LIN {X 0,Y 162.947,Z 318.354,A -85,B 0,C 180,E1 -26149.316,E2 -26149.316} C_VEL
LIN {X 0,Y 160.484,Z 333.964,A -85,B 0,C 180,E1 -26150.172,E2 -26150.172} C_VEL
LIN {X 0,Y 157.007,Z 349.23,A -85,B 0,C 180,E1 -26151.399,E2 -26151.399} C_VEL
LIN {X 0,Y 152.992,Z 362.96,A -85,B 0,C 180,E1 -26152.919,E2 -26152.919} C_VEL
LIN {X 0,Y 148.184,Z 376.471,A -85,B 0,C 180,E1 -26154.895,E2 -26154.895} C_VEL
LIN {X 0,Y 142.969,Z 388.947,A -85,B 0,C 180,E1 -26157.265,E2 -26157.265} C_VEL
LIN {X 0,Y 137.361,Z 400.576,A -85,B 0,C 180,E1 -26160.074,E2 -26160.074} C_VEL
LIN {X 0,Y 131.045,Z 412.295,A -85,B 0,C 180,E1 -26163.738,E2 -26163.738} C_VEL
LIN {X 0,Y 125.325,Z 422.137,A -85,B 0,C 180,E1 -26167.756,E2 -26167.756} C_VEL
LIN {X 0,Y 119.407,Z 431.78,A -85,B 0,C 180,E1 -26172.884,E2 -26172.884} C_VEL
LIN {X 0,Y 115.037,Z 438.966,A -85,B 0,C 180,E1 -26177.828,E2 -26177.828} C_VEL
LIN {X 0,Y 110.501,Z 446.462,A -85,B 0,C 180,E1 -26184.524,E2 -26184.524} C_VEL
LIN {X 0,Y 107.298,Z 452.585,A -85,B 0,C 180,E1 -26191.875,E2 -26191.875} C_VEL
LIN {X 0,Y 105.639,Z 456.228,A -85,B 0,C 180,E1 -26197.645,E2 -26197.645} C_VEL
LIN {X 0,Y 104.586,Z 459.955,A -85,B 0,C 180,E1 -26205.591,E2 -26205.591} C_VEL
LIN {X 0,Y 104.541,Z 461.374,A -85,B 0,C 180,E1 -26209.743,E2 -26209.743} C_VEL
LIN {X 0,Y 105.346,Z 463.187,A -85,B 0,C 180,E1 -26217.838,E2 -26217.838} C_VEL
LIN {X 0,Y 107.662,Z 463.763,A -85,B 0,C 180,E1 -26225.978,E2 -26225.978} C_VEL
LIN {X 0,Y 111.789,Z 463.039,A -85,B 0,C 180,E1 -26233.751,E2 -26233.751} C_VEL
LIN {X 0,Y 117.628,Z 460.978,A -85,B 0,C 180,E1 -26240.959,E2 -26240.959} C_VEL
LIN {X 0,Y 125.074,Z 457.514,A -85,B 0,C 180,E1 -26247.441,E2 -26247.441} C_VEL
LIN {X 0,Y 133.883,Z 452.565,A -85,B 0,C 180,E1 -26253.173,E2 -26253.173} C_VEL
LIN {X 0,Y 143.854,Z 445.982,A -85,B 0,C 180,E1 -26258.161,E2 -26258.161} C_VEL
LIN {X 0,Y 152.435,Z 439.533,A -85,B 0,C 180,E1 -26261.583,E2 -26261.583} C_VEL
LIN {X 0,Y 162.624,Z 430.726,A -85,B 0,C 180,E1 -26264.971,E2 -26264.971} C_VEL
LIN {X 0,Y 172.579,Z 420.723,A -85,B 0,C 180,E1 -26267.781,E2 -26267.781} C_VEL
LIN {X 0,Y 181.957,Z 409.798,A -85,B 0,C 180,E1 -26270.035,E2 -26270.035} C_VEL
LIN {X 0,Y 190.529,Z 398.113,A -85,B 0,C 180,E1 -26271.871,E2 -26271.871} C_VEL
LIN {X 0,Y 198.109,Z 385.919,A -85,B 0,C 180,E1 -26273.364,E2 -26273.364} C_VEL
LIN {X 0,Y 204.736,Z 373.274,A -85,B 0,C 180,E1 -26274.55,E2 -26274.55} C_VEL
LIN {X 0,Y 211.024,Z 358.642,A -85,B 0,C 180,E1 -26275.59,E2 -26275.59} C_VEL
LIN {X 0,Y 215.218,Z 346.337,A -85,B 0,C 180,E1 -26276.255,E2 -26276.255} C_VEL
LIN {X 0,Y 219.141,Z 331.367,A -85,B 0,C 180,E1 -26276.858,E2 -26276.858} C_VEL
LIN {X 0,Y 221.825,Z 316.289,A -85,B 0,C 180,E1 -26277.276,E2 -26277.276} C_VEL
LIN {X 0,Y 224.175,Z 295.698,A -85,B 0,C 180,E1 -26277.764,E2 -26277.764} C_VEL
LIN {X 0,Y 222.622,Z 291.518,A -85,B 0,C 180,E1 -26280.578,E2 -26280.578} C_VEL
LIN {X 0,Y 221.196,Z 287.861,A -85,B 0,C 180,E1 -26284.477,E2 -26284.477} C_VEL
LIN {X 0,Y 220.426,Z 286.824,A -85,B 0,C 180,E1 -26289.172,E2 -26289.172} C_VEL
LIN {X 0,Y 221.19,Z 288.234,A -85,B 0,C 180,E1 -26294.297,E2 -26294.297} C_VEL
LIN {X 0,Y 222.327,Z 291.545,A -85,B 0,C 180,E1 -26297.604,E2 -26297.604} C_VEL
LIN {X 0,Y 223.799,Z 296.565,A -85,B 0,C 180,E1 -26300.586,E2 -26300.586} C_VEL
LIN {X 0,Y 224.016,Z 297.417,A -85,B 0,C 180,E1 -26300.965,E2 -26300.965} C_VEL
LIN {X 0,Y 221.746,Z 317.672,A -85,B 0,C 180,E1 -26301.455,E2 -26301.455} C_VEL
LIN {X 0,Y 219.086,Z 333.204,A -85,B 0,C 180,E1 -26301.867,E2 -26301.867} C_VEL
LIN {X 0,Y 215.269,Z 347.941,A -85,B 0,C 180,E1 -26302.373,E2 -26302.373} C_VEL
LIN {X 0,Y 210.855,Z 360.923,A -85,B 0,C 180,E1 -26302.963,E2 -26302.963} C_VEL
LIN {X 0,Y 204.602,Z 375.459,A -85,B 0,C 180,E1 -26303.858,E2 -26303.858} C_VEL
LIN {X 0,Y 197.67,Z 388.649,A -85,B 0,C 180,E1 -26304.957,E2 -26304.957} C_VEL
LIN {X 0,Y 189.342,Z 401.874,A -85,B 0,C 180,E1 -26306.432,E2 -26306.432} C_VEL
LIN {X 0,Y 182.696,Z 411,A -85,B 0,C 180,E1 -26307.778,E2 -26307.778} C_VEL
LIN {X 0,Y 174.076,Z 421.494,A -85,B 0,C 180,E1 -26309.772,E2 -26309.772} C_VEL
LIN {X 0,Y 165.563,Z 430.476,A -85,B 0,C 180,E1 -26311.9,E2 -26311.9} C_VEL
LIN {X 0,Y 156.09,Z 439.328,A -85,B 0,C 180,E1 -26314.745,E2 -26314.745} C_VEL
LIN {X 0,Y 146.989,Z 446.713,A -85,B 0,C 180,E1 -26317.917,E2 -26317.917} C_VEL
LIN {X 0,Y 139.667,Z 452.041,A -85,B 0,C 180,E1 -26320.994,E2 -26320.994} C_VEL
LIN {X 0,Y 130.857,Z 457.904,A -85,B 0,C 180,E1 -26325.719,E2 -26325.719} C_VEL
LIN {X 0,Y 122.947,Z 462.477,A -85,B 0,C 180,E1 -26331.041,E2 -26331.041} C_VEL
LIN {X 0,Y 116.264,Z 465.806,A -85,B 0,C 180,E1 -26337.043,E2 -26337.043} C_VEL
LIN {X 0,Y 111.028,Z 467.995,A -85,B 0,C 180,E1 -26343.7,E2 -26343.7} C_VEL
LIN {X 0,Y 107.414,Z 469.101,A -85,B 0,C 180,E1 -26350.906,E2 -26350.906} C_VEL
LIN {X 0,Y 105.512,Z 469.138,A -85,B 0,C 180,E1 -26358.475,E2 -26358.475} C_VEL
LIN {X 0,Y 105.017,Z 468.005,A -85,B 0,C 180,E1 -26366.164,E2 -26366.164} C_VEL
LIN {X 0,Y 105.227,Z 467.01,A -85,B 0,C 180,E1 -26370.002,E2 -26370.002} C_VEL
LIN {X 0,Y 105.077,Z 466.112,A -85,B 0,C 180,E1 -26372.599,E2 -26372.599} C_VEL
LIN {X 0,Y 104.753,Z 465.346,A -85,B 0,C 180,E1 -26374.699,E2 -26374.699} C_VEL
LIN {X 0,Y 103.497,Z 463.984,A -85,B 0,C 180,E1 -26377.803,E2 -26377.803} C_VEL
LIN {X 0,Y 100.091,Z 460.077,A -85,B 0,C 180,E1 -26385.125,E2 -26385.125} C_VEL
LIN {X 0,Y 99.855,Z 458.028,A -85,B 0,C 180,E1 -26388.335,E2 -26388.335} C_VEL
LIN {X 0,Y 100.106,Z 457.282,A -85,B 0,C 180,E1 -26389.384,E2 -26389.384} C_VEL
LIN {X 0,Y 103.055,Z 451.741,A -85,B 0,C 180,E1 -26396.315,E2 -26396.315} C_VEL
LIN {X 0,Y 107.909,Z 443.902,A -85,B 0,C 180,E1 -26403.616,E2 -26403.616} C_VEL
LIN {X 0,Y 113.461,Z 435.505,A -85,B 0,C 180,E1 -26409.415,E2 -26409.415} C_VEL
LIN {X 0,Y 119.894,Z 425.346,A -85,B 0,C 180,E1 -26414.704,E2 -26414.704} C_VEL
LIN {X 0,Y 126.204,Z 414.925,A -85,B 0,C 180,E1 -26418.747,E2 -26418.747} C_VEL
LIN {X 0,Y 132.977,Z 402.455,A -85,B 0,C 180,E1 -26422.447,E2 -26422.447} C_VEL
LIN {X 0,Y 139.15,Z 389.961,A -85,B 0,C 180,E1 -26425.161,E2 -26425.161} C_VEL
LIN {X 0,Y 145.14,Z 375.71,A -85,B 0,C 180,E1 -26427.507,E2 -26427.507} C_VEL
LIN {X 0,Y 150.15,Z 361.027,A -85,B 0,C 180,E1 -26429.327,E2 -26429.327} C_VEL
LIN {X 0,Y 154.269,Z 346.233,A -85,B 0,C 180,E1 -26430.61,E2 -26430.61} C_VEL
LIN {X 0,Y 157.337,Z 330.894,A -85,B 0,C 180,E1 -26431.574,E2 -26431.574} C_VEL
LIN {X 0,Y 159.384,Z 314.642,A -85,B 0,C 180,E1 -26432.232,E2 -26432.232} C_VEL
LIN {X 0,Y 164.239,Z 261.106,A -85,B 0,C 180,E1 -26433.98,E2 -26433.98} C_VEL
LIN {X 0,Y 160.374,Z 249.054,A -85,B 0,C 180,E1 -26437.113,E2 -26437.113} C_VEL
LIN {X 0,Y 157.851,Z 243.64,A -85,B 0,C 180,E1 -26439.135,E2 -26439.135} C_VEL
LIN {X 0,Y 154.336,Z 236.992,A -85,B 0,C 180,E1 -26442.213,E2 -26442.213} C_VEL
LIN {X 0,Y 150.77,Z 230.752,A -85,B 0,C 180,E1 -26445.836,E2 -26445.836} C_VEL
LIN {X 0,Y 148.532,Z 226.927,A -85,B 0,C 180,E1 -26448.51,E2 -26448.51} C_VEL
LIN {X 0,Y 146.901,Z 224.205,A -85,B 0,C 180,E1 -26450.747,E2 -26450.747} C_VEL
LIN {X 0,Y 144.473,Z 220.156,A -85,B 0,C 180,E1 -26454.7,E2 -26454.7} C_VEL
LIN {X 0,Y 142.281,Z 216.757,A -85,B 0,C 180,E1 -26459.526,E2 -26459.526} C_VEL
LIN {X 0,Y 141.888,Z 215.561,A -85,B 0,C 180,E1 -26460.888,E2 -26460.888} C_VEL
LIN {X 0,Y 140.44,Z 214.72,A -85,B 0,C 180,E1 -26468.636,E2 -26468.636} C_VEL
LIN {X 0,Y 141.644,Z 216.006,A -85,B 0,C 180,E1 -26478.067,E2 -26478.067} C_VEL
LIN {X 0,Y 142.299,Z 217.543,A -85,B 0,C 180,E1 -26480.227,E2 -26480.227} C_VEL
LIN {X 0,Y 144.869,Z 221.173,A -85,B 0,C 180,E1 -26485.565,E2 -26485.565} C_VEL
LIN {X 0,Y 147.719,Z 225.741,A -85,B 0,C 180,E1 -26489.909,E2 -26489.909} C_VEL
LIN {X 0,Y 150.199,Z 229.95,A -85,B 0,C 180,E1 -26493.014,E2 -26493.014} C_VEL
LIN {X 0,Y 153.362,Z 235.256,A -85,B 0,C 180,E1 -26496.335,E2 -26496.335} C_VEL
LIN {X 0,Y 158.282,Z 244.468,A -85,B 0,C 180,E1 -26500.696,E2 -26500.696} C_VEL
LIN {X 0,Y 163.058,Z 254.709,A -85,B 0,C 180,E1 -26504.353,E2 -26504.353} C_VEL
LIN {X 0,Y 164.466,Z 258.317,A -85,B 0,C 180,E1 -26505.39,E2 -26505.39} C_VEL
LIN {X 0,Y 158.621,Z 318.896,A -85,B 0,C 180,E1 -26507.314,E2 -26507.314} C_VEL
LIN {X 0,Y 156.073,Z 334.383,A -85,B 0,C 180,E1 -26508.162,E2 -26508.162} C_VEL
LIN {X 0,Y 152.499,Z 349.571,A -85,B 0,C 180,E1 -26509.385,E2 -26509.385} C_VEL
LIN {X 0,Y 148.01,Z 364.208,A -85,B 0,C 180,E1 -26511.011,E2 -26511.011} C_VEL
LIN {X 0,Y 143.019,Z 377.559,A -85,B 0,C 180,E1 -26512.987,E2 -26512.987} C_VEL
LIN {X 0,Y 137.012,Z 391.148,A -85,B 0,C 180,E1 -26515.649,E2 -26515.649} C_VEL
LIN {X 0,Y 130.631,Z 403.517,A -85,B 0,C 180,E1 -26518.812,E2 -26518.812} C_VEL
LIN {X 0,Y 123.656,Z 415.61,A -85,B 0,C 180,E1 -26522.954,E2 -26522.954} C_VEL
LIN {X 0,Y 117.811,Z 425.011,A -85,B 0,C 180,E1 -26527.183,E2 -26527.183} C_VEL
LIN {X 0,Y 111.83,Z 434.197,A -85,B 0,C 180,E1 -26532.63,E2 -26532.63} C_VEL
LIN {X 0,Y 106.791,Z 441.825,A -85,B 0,C 180,E1 -26538.612,E2 -26538.612} C_VEL
LIN {X 0,Y 102.362,Z 448.961,A -85,B 0,C 180,E1 -26546.062,E2 -26546.062} C_VEL
LIN {X 0,Y 99.423,Z 454.572,A -85,B 0,C 180,E1 -26554.052,E2 -26554.052} C_VEL
LIN {X 0,Y 97.71,Z 458.826,A -85,B 0,C 180,E1 -26562.46,E2 -26562.46} C_VEL
LIN {X 0,Y 97.454,Z 461.574,A -85,B 0,C 180,E1 -26570.358,E2 -26570.358} C_VEL
LIN {X 0,Y 97.844,Z 462.804,A -85,B 0,C 180,E1 -26575.528,E2 -26575.528} C_VEL
LIN {X 0,Y 99.81,Z 463.886,A -85,B 0,C 180,E1 -26584.283,E2 -26584.283} C_VEL
LIN {X 0,Y 103.648,Z 463.679,A -85,B 0,C 180,E1 -26592.69,E2 -26592.69} C_VEL
LIN {X 0,Y 109.367,Z 462.158,A -85,B 0,C 180,E1 -26600.453,E2 -26600.453} C_VEL
LIN {X 0,Y 116.758,Z 459.274,A -85,B 0,C 180,E1 -26607.424,E2 -26607.424} C_VEL
LIN {X 0,Y 125.628,Z 454.943,A -85,B 0,C 180,E1 -26613.517,E2 -26613.517} C_VEL
LIN {X 0,Y 135.712,Z 449.048,A -85,B 0,C 180,E1 -26618.769,E2 -26618.769} C_VEL
LIN {X 0,Y 145.355,Z 442.484,A -85,B 0,C 180,E1 -26622.728,E2 -26622.728} C_VEL
LIN {X 0,Y 155.63,Z 434.4,A -85,B 0,C 180,E1 -26626.141,E2 -26626.141} C_VEL
LIN {X 0,Y 164.815,Z 426.083,A -85,B 0,C 180,E1 -26628.738,E2 -26628.738} C_VEL
LIN {X 0,Y 174.502,Z 415.934,A -85,B 0,C 180,E1 -26631.105,E2 -26631.105} C_VEL
LIN {X 0,Y 184.056,Z 404.264,A -85,B 0,C 180,E1 -26633.109,E2 -26633.109} C_VEL
LIN {X 0,Y 192.337,Z 392.315,A -85,B 0,C 180,E1 -26634.686,E2 -26634.686} C_VEL
LIN {X 0,Y 199.672,Z 379.769,A -85,B 0,C 180,E1 -26635.962,E2 -26635.962} C_VEL
LIN {X 0,Y 205.86,Z 367.093,A -85,B 0,C 180,E1 -26636.944,E2 -26636.944} C_VEL
LIN {X 0,Y 211,Z 354.174,A -85,B 0,C 180,E1 -26637.753,E2 -26637.753} C_VEL
LIN {X 0,Y 215.847,Z 338.673,A -85,B 0,C 180,E1 -26638.413,E2 -26638.413} C_VEL
LIN {X 0,Y 219.226,Z 323.398,A -85,B 0,C 180,E1 -26638.895,E2 -26638.895} C_VEL
LIN {X 0,Y 222.037,Z 302.205,A -85,B 0,C 180,E1 -26639.38,E2 -26639.38} C_VEL
LIN {X 0,Y 222.2,Z 300.533,A -85,B 0,C 180,E1 -26639.455,E2 -26639.455} C_VEL
LIN {X 0,Y 221.192,Z 297.74,A -85,B 0,C 180,E1 -26641.656,E2 -26641.656} C_VEL
LIN {X 0,Y 220.189,Z 294.827,A -85,B 0,C 180,E1 -26644.821,E2 -26644.821} C_VEL
LIN {X 0,Y 219.525,Z 293.886,A -85,B 0,C 180,E1 -26649.21,E2 -26649.21} C_VEL
LIN {X 0,Y 220.207,Z 295.224,A -85,B 0,C 180,E1 -26654.04,E2 -26654.04} C_VEL
LIN {X 0,Y 221.155,Z 298.273,A -85,B 0,C 180,E1 -26657.064,E2 -26657.064} C_VEL
LIN {X 0,Y 222.091,Z 301.931,A -85,B 0,C 180,E1 -26659.313,E2 -26659.313} C_VEL
LIN {X 0,Y 219.112,Z 325.05,A -85,B 0,C 180,E1 -26659.828,E2 -26659.828} C_VEL
LIN {X 0,Y 215.67,Z 340.76,A -85,B 0,C 180,E1 -26660.28,E2 -26660.28} C_VEL
LIN {X 0,Y 210.999,Z 355.769,A -85,B 0,C 180,E1 -26660.843,E2 -26660.843} C_VEL
LIN {X 0,Y 205.037,Z 370.484,A -85,B 0,C 180,E1 -26661.604,E2 -26661.604} C_VEL
LIN {X 0,Y 197.956,Z 384.544,A -85,B 0,C 180,E1 -26662.622,E2 -26662.622} C_VEL
LIN {X 0,Y 190.179,Z 397.334,A -85,B 0,C 180,E1 -26663.849,E2 -26663.849} C_VEL
LIN {X 0,Y 182.334,Z 408.337,A -85,B 0,C 180,E1 -26665.211,E2 -26665.211} C_VEL
LIN {X 0,Y 173.589,Z 419.061,A -85,B 0,C 180,E1 -26667.04,E2 -26667.04} C_VEL
LIN {X 0,Y 163.377,Z 429.744,A -85,B 0,C 180,E1 -26669.416,E2 -26669.416} C_VEL
LIN {X 0,Y 153.549,Z 438.668,A -85,B 0,C 180,E1 -26672.141,E2 -26672.141} C_VEL
LIN {X 0,Y 142.746,Z 447.11,A -85,B 0,C 180,E1 -26675.674,E2 -26675.674} C_VEL
LIN {X 0,Y 132.706,Z 453.923,A -85,B 0,C 180,E1 -26679.835,E2 -26679.835} C_VEL
LIN {X 0,Y 123.636,Z 459.316,A -85,B 0,C 180,E1 -26684.722,E2 -26684.722} C_VEL
LIN {X 0,Y 117.479,Z 462.551,A -85,B 0,C 180,E1 -26688.849,E2 -26688.849} C_VEL
LIN {X 0,Y 110.324,Z 465.814,A -85,B 0,C 180,E1 -26695.019,E2 -26695.019} C_VEL
LIN {X 0,Y 104.657,Z 467.905,A -85,B 0,C 180,E1 -26701.963,E2 -26701.963} C_VEL
LIN {X 0,Y 100.686,Z 468.923,A -85,B 0,C 180,E1 -26709.575,E2 -26709.575} C_VEL
LIN {X 0,Y 98.543,Z 468.873,A -85,B 0,C 180,E1 -26717.647,E2 -26717.647} C_VEL
LIN {X 0,Y 97.92,Z 467.695,A -85,B 0,C 180,E1 -26725.886,E2 -26725.886} C_VEL
LIN {X 0,Y 98.138,Z 466.656,A -85,B 0,C 180,E1 -26730.002,E2 -26730.002} C_VEL
LIN {X 0,Y 97.993,Z 465.285,A -85,B 0,C 180,E1 -26734.114,E2 -26734.114} C_VEL
LIN {X 0,Y 98.512,Z 461.576,A -85,B 0,C 180,E1 -26742.36,E2 -26742.36} C_VEL
LIN {X 0,Y 100.106,Z 457.282,A -85,B 0,C 180,E1 -26749.384,E2 -26749.384} C_VEL
LIN {X 0,Y 100.588,Z 455.059,A -85,B 0,C 180,E1 -26752.484,E2 -26752.484} C_VEL
LIN {X 0,Y 100.113,Z 450.987,A -85,B 0,C 180,E1 -26757.659,E2 -26757.659} C_VEL
LIN {X 0,Y 100.279,Z 446.507,A -85,B 0,C 180,E1 -26762.738,E2 -26762.738} C_VEL
LIN {X 0,Y 101.703,Z 443.492,A -85,B 0,C 180,E1 -26765.515,E2 -26765.515} C_VEL
LIN {X 0,Y 107.999,Z 434.564,A -85,B 0,C 180,E1 -26771.839,E2 -26771.839} C_VEL
LIN {X 0,Y 113.836,Z 425.841,A -85,B 0,C 180,E1 -26776.506,E2 -26776.506} C_VEL
LIN {X 0,Y 120.427,Z 415.547,A -85,B 0,C 180,E1 -26780.65,E2 -26780.65} C_VEL
LIN {X 0,Y 126.879,Z 404.343,A -85,B 0,C 180,E1 -26784.108,E2 -26784.108} C_VEL
LIN {X 0,Y 133.246,Z 392.275,A -85,B 0,C 180,E1 -26786.861,E2 -26786.861} C_VEL
LIN {X 0,Y 138.51,Z 380.778,A -85,B 0,C 180,E1 -26788.899,E2 -26788.899} C_VEL
LIN {X 0,Y 143.867,Z 366.706,A -85,B 0,C 180,E1 -26790.85,E2 -26790.85} C_VEL
LIN {X 0,Y 148.046,Z 353.721,A -85,B 0,C 180,E1 -26792.151,E2 -26792.151} C_VEL
LIN {X 0,Y 151.72,Z 338.711,A -85,B 0,C 180,E1 -26793.274,E2 -26793.274} C_VEL
LIN {X 0,Y 154.404,Z 323.324,A -85,B 0,C 180,E1 -26794.024,E2 -26794.024} C_VEL
LIN {X 0,Y 160.176,Z 263.515,A -85,B 0,C 180,E1 -26795.985,E2 -26795.985} C_VEL
LIN {X 0,Y 156.681,Z 252.456,A -85,B 0,C 180,E1 -26799.058,E2 -26799.058} C_VEL
LIN {X 0,Y 152.347,Z 243.572,A -85,B 0,C 180,E1 -26803.018,E2 -26803.018} C_VEL
LIN {X 0,Y 148.714,Z 236.88,A -85,B 0,C 180,E1 -26806.966,E2 -26806.966} C_VEL
LIN {X 0,Y 146.507,Z 232.886,A -85,B 0,C 180,E1 -26809.844,E2 -26809.844} C_VEL
LIN {X 0,Y 145.297,Z 230.723,A -85,B 0,C 180,E1 -26811.658,E2 -26811.658} C_VEL
LIN {X 0,Y 142.89,Z 226.63,A -85,B 0,C 180,E1 -26815.861,E2 -26815.861} C_VEL
LIN {X 0,Y 140.991,Z 223.16,A -85,B 0,C 180,E1 -26820.671,E2 -26820.671} C_VEL
LIN {X 0,Y 140.643,Z 222.434,A -85,B 0,C 180,E1 -26821.931,E2 -26821.931} C_VEL
LIN {X 0,Y 139.526,Z 221.864,A -85,B 0,C 180,E1 -26830.162,E2 -26830.162} C_VEL
LIN {X 0,Y 140.755,Z 223.236,A -85,B 0,C 180,E1 -26838.185,E2 -26838.185} C_VEL
LIN {X 0,Y 142.628,Z 226.799,A -85,B 0,C 180,E1 -26843.218,E2 -26843.218} C_VEL
LIN {X 0,Y 143.409,Z 227.797,A -85,B 0,C 180,E1 -26844.697,E2 -26844.697} C_VEL
LIN {X 0,Y 146.029,Z 232.223,A -85,B 0,C 180,E1 -26848.964,E2 -26848.964} C_VEL
LIN {X 0,Y 148.528,Z 236.692,A -85,B 0,C 180,E1 -26852.302,E2 -26852.302} C_VEL
LIN {X 0,Y 151.504,Z 242.08,A -85,B 0,C 180,E1 -26855.617,E2 -26855.617} C_VEL
LIN {X 0,Y 155.718,Z 250.393,A -85,B 0,C 180,E1 -26859.595,E2 -26859.595} C_VEL
LIN {X 0,Y 160.217,Z 260.619,A -85,B 0,C 180,E1 -26863.27,E2 -26863.27} C_VEL
LIN {X 0,Y 160.186,Z 262.86,A -85,B 0,C 180,E1 -26863.442,E2 -26863.442} C_VEL
LIN {X 0,Y 154.518,Z 319.309,A -85,B 0,C 180,E1 -26865.199,E2 -26865.199} C_VEL
LIN {X 0,Y 151.872,Z 334.788,A -85,B 0,C 180,E1 -26866.04,E2 -26866.04} C_VEL
LIN {X 0,Y 148.172,Z 349.925,A -85,B 0,C 180,E1 -26867.244,E2 -26867.244} C_VEL
LIN {X 0,Y 143.869,Z 363.61,A -85,B 0,C 180,E1 -26868.739,E2 -26868.739} C_VEL
LIN {X 0,Y 138.692,Z 377.075,A -85,B 0,C 180,E1 -26870.696,E2 -26870.696} C_VEL
LIN {X 0,Y 133.046,Z 389.515,A -85,B 0,C 180,E1 -26873.066,E2 -26873.066} C_VEL
LIN {X 0,Y 127.404,Z 400.28,A -85,B 0,C 180,E1 -26875.675,E2 -26875.675} C_VEL
LIN {X 0,Y 120.584,Z 411.909,A -85,B 0,C 180,E1 -26879.336,E2 -26879.336} C_VEL
LIN {X 0,Y 114.193,Z 421.883,A -85,B 0,C 180,E1 -26883.498,E2 -26883.498} C_VEL
LIN {X 0,Y 107.547,Z 431.631,A -85,B 0,C 180,E1 -26888.934,E2 -26888.934} C_VEL
LIN {X 0,Y 101.82,Z 439.845,A -85,B 0,C 180,E1 -26895.098,E2 -26895.098} C_VEL
LIN {X 0,Y 97.28,Z 446.499,A -85,B 0,C 180,E1 -26901.691,E2 -26901.691} C_VEL
LIN {X 0,Y 93.494,Z 452.705,A -85,B 0,C 180,E1 -26909.998,E2 -26909.998} C_VEL
LIN {X 0,Y 91.819,Z 455.931,A -85,B 0,C 180,E1 -26915.685,E2 -26915.685} C_VEL
LIN {X 0,Y 90.491,Z 459.4,A -85,B 0,C 180,E1 -26923.472,E2 -26923.472} C_VEL
LIN {X 0,Y 90.369,Z 461.769,A -85,B 0,C 180,E1 -26931.049,E2 -26931.049} C_VEL
LIN {X 0,Y 91.003,Z 463.187,A -85,B 0,C 180,E1 -26937.603,E2 -26937.603} C_VEL
LIN {X 0,Y 93.523,Z 464.135,A -85,B 0,C 180,E1 -26946.952,E2 -26946.952} C_VEL
LIN {X 0,Y 98.056,Z 463.797,A -85,B 0,C 180,E1 -26955.783,E2 -26955.783} C_VEL
LIN {X 0,Y 104.544,Z 462.146,A -85,B 0,C 180,E1 -26963.773,E2 -26963.773} C_VEL
LIN {X 0,Y 112.726,Z 459.125,A -85,B 0,C 180,E1 -26970.788,E2 -26970.788} C_VEL
LIN {X 0,Y 122.339,Z 454.653,A -85,B 0,C 180,E1 -26976.8,E2 -26976.8} C_VEL
LIN {X 0,Y 133.076,Z 448.607,A -85,B 0,C 180,E1 -26981.916,E2 -26981.916} C_VEL
LIN {X 0,Y 143.735,Z 441.535,A -85,B 0,C 180,E1 -26985.848,E2 -26985.848} C_VEL
LIN {X 0,Y 153.96,Z 433.619,A -85,B 0,C 180,E1 -26988.938,E2 -26988.938} C_VEL
LIN {X 0,Y 163.477,Z 425.103,A -85,B 0,C 180,E1 -26991.407,E2 -26991.407} C_VEL
LIN {X 0,Y 173.273,Z 414.976,A -85,B 0,C 180,E1 -26993.573,E2 -26993.573} C_VEL
LIN {X 0,Y 182.452,Z 403.917,A -85,B 0,C 180,E1 -26995.333,E2 -26995.333} C_VEL
LIN {X 0,Y 190.925,Z 391.876,A -85,B 0,C 180,E1 -26996.827,E2 -26996.827} C_VEL
LIN {X 0,Y 199.057,Z 378.052,A -85,B 0,C 180,E1 -26998.119,E2 -26998.119} C_VEL
LIN {X 0,Y 205.594,Z 364.537,A -85,B 0,C 180,E1 -26999.065,E2 -26999.065} C_VEL
LIN {X 0,Y 211.246,Z 349.794,A -85,B 0,C 180,E1 -26999.86,E2 -26999.86} C_VEL
LIN {X 0,Y 215.751,Z 334.209,A -85,B 0,C 180,E1 -27000.437,E2 -27000.437} C_VEL
LIN {X 0,Y 218.769,Z 319.005,A -85,B 0,C 180,E1 -27000.848,E2 -27000.848} C_VEL
LIN {X 0,Y 220.476,Z 305.596,A -85,B 0,C 180,E1 -27001.132,E2 -27001.132} C_VEL
LIN {X 0,Y 219.187,Z 301.783,A -85,B 0,C 180,E1 -27005.181,E2 -27005.181} C_VEL
LIN {X 0,Y 218.626,Z 300.947,A -85,B 0,C 180,E1 -27009.249,E2 -27009.249} C_VEL
LIN {X 0,Y 219.215,Z 302.209,A -85,B 0,C 180,E1 -27013.74,E2 -27013.74} C_VEL
LIN {X 0,Y 220.017,Z 304.976,A -85,B 0,C 180,E1 -27016.541,E2 -27016.541} C_VEL
LIN {X 0,Y 220.377,Z 306.541,A -85,B 0,C 180,E1 -27017.57,E2 -27017.57} C_VEL
LIN {X 0,Y 217.642,Z 326.275,A -85,B 0,C 180,E1 -27018.026,E2 -27018.026} C_VEL
LIN {X 0,Y 214.133,Z 341.502,A -85,B 0,C 180,E1 -27018.442,E2 -27018.442} C_VEL
LIN {X 0,Y 209.459,Z 356.062,A -85,B 0,C 180,E1 -27018.96,E2 -27018.96} C_VEL
LIN {X 0,Y 203.38,Z 370.687,A -85,B 0,C 180,E1 -27019.671,E2 -27019.671} C_VEL
LIN {X 0,Y 196.166,Z 384.641,A -85,B 0,C 180,E1 -27020.615,E2 -27020.615} C_VEL
LIN {X 0,Y 188.244,Z 397.364,A -85,B 0,C 180,E1 -27021.769,E2 -27021.769} C_VEL
LIN {X 0,Y 179.594,Z 409.116,A -85,B 0,C 180,E1 -27023.154,E2 -27023.154} C_VEL
LIN {X 0,Y 170.506,Z 419.829,A -85,B 0,C 180,E1 -27024.934,E2 -27024.934} C_VEL
LIN {X 0,Y 160.032,Z 430.349,A -85,B 0,C 180,E1 -27027.216,E2 -27027.216} C_VEL
LIN {X 0,Y 149.892,Z 439.157,A -85,B 0,C 180,E1 -27029.843,E2 -27029.843} C_VEL
LIN {X 0,Y 138.719,Z 447.461,A -85,B 0,C 180,E1 -27033.287,E2 -27033.287} C_VEL
LIN {X 0,Y 128.25,Z 454.181,A -85,B 0,C 180,E1 -27037.385,E2 -27037.385} C_VEL
LIN {X 0,Y 118.729,Z 459.49,A -85,B 0,C 180,E1 -27042.277,E2 -27042.277} C_VEL
LIN {X 0,Y 112.189,Z 462.619,A -85,B 0,C 180,E1 -27046.444,E2 -27046.444} C_VEL
LIN {X 0,Y 104.545,Z 465.811,A -85,B 0,C 180,E1 -27052.771,E2 -27052.771} C_VEL
LIN {X 0,Y 98.382,Z 467.823,A -85,B 0,C 180,E1 -27059.998,E2 -27059.998} C_VEL
LIN {X 0,Y 94.025,Z 468.745,A -85,B 0,C 180,E1 -27068.056,E2 -27068.056} C_VEL
LIN {X 0,Y 91.574,Z 468.605,A -85,B 0,C 180,E1 -27076.691,E2 -27076.691} C_VEL
LIN {X 0,Y 90.846,Z 467.371,A -85,B 0,C 180,E1 -27085.565,E2 -27085.565} C_VEL
LIN {X 0,Y 91.04,Z 466.302,A -85,B 0,C 180,E1 -27090.002,E2 -27090.002} C_VEL
LIN {X 0,Y 90.899,Z 464.885,A -85,B 0,C 180,E1 -27094.436,E2 -27094.436} C_VEL
LIN {X 0,Y 91.54,Z 461.079,A -85,B 0,C 180,E1 -27103.318,E2 -27103.318} C_VEL
LIN {X 0,Y 93.786,Z 455.892,A -85,B 0,C 180,E1 -27112.007,E2 -27112.007} C_VEL
LIN {X 0,Y 97.811,Z 449.19,A -85,B 0,C 180,E1 -27120.199,E2 -27120.199} C_VEL
LIN {X 0,Y 101.703,Z 443.492,A -85,B 0,C 180,E1 -27125.515,E2 -27125.515} C_VEL
LIN {X 0,Y 103.31,Z 440.352,A -85,B 0,C 180,E1 -27128.15,E2 -27128.15} C_VEL
LIN {X 0,Y 104.717,Z 434.939,A -85,B 0,C 180,E1 -27132.646,E2 -27132.646} C_VEL
LIN {X 0,Y 106.515,Z 429.077,A -85,B 0,C 180,E1 -27136.9,E2 -27136.9} C_VEL
LIN {X 0,Y 108.648,Z 425.222,A -85,B 0,C 180,E1 -27139.048,E2 -27139.048} C_VEL
LIN {X 0,Y 115.966,Z 414.31,A -85,B 0,C 180,E1 -27143.421,E2 -27143.421} C_VEL
LIN {X 0,Y 123.406,Z 401.772,A -85,B 0,C 180,E1 -27147.145,E2 -27147.145} C_VEL
LIN {X 0,Y 130.086,Z 389.223,A -85,B 0,C 180,E1 -27149.819,E2 -27149.819} C_VEL
LIN {X 0,Y 136.358,Z 375.272,A -85,B 0,C 180,E1 -27152.051,E2 -27152.051} C_VEL
LIN {X 0,Y 141.531,Z 361.146,A -85,B 0,C 180,E1 -27153.76,E2 -27153.76} C_VEL
LIN {X 0,Y 145.912,Z 346.519,A -85,B 0,C 180,E1 -27154.978,E2 -27154.978} C_VEL
LIN {X 0,Y 149.302,Z 330.674,A -85,B 0,C 180,E1 -27155.944,E2 -27155.944} C_VEL
LIN {X 0,Y 151.418,Z 315.134,A -85,B 0,C 180,E1 -27156.556,E2 -27156.556} C_VEL
LIN {X 0,Y 156.234,Z 265.975,A -85,B 0,C 180,E1 -27158.087,E2 -27158.087} C_VEL
LIN {X 0,Y 153.542,Z 257.126,A -85,B 0,C 180,E1 -27160.707,E2 -27160.707} C_VEL
LIN {X 0,Y 149.749,Z 248.945,A -85,B 0,C 180,E1 -27164.52,E2 -27164.52} C_VEL
LIN {X 0,Y 146.49,Z 242.527,A -85,B 0,C 180,E1 -27168.432,E2 -27168.432} C_VEL
LIN {X 0,Y 143.885,Z 237.458,A -85,B 0,C 180,E1 -27172.327,E2 -27172.327} C_VEL
LIN {X 0,Y 141.631,Z 233.444,A -85,B 0,C 180,E1 -27176.491,E2 -27176.491} C_VEL
LIN {X 0,Y 139.827,Z 229.832,A -85,B 0,C 180,E1 -27181.525,E2 -27181.525} C_VEL
LIN {X 0,Y 139.469,Z 229.348,A -85,B 0,C 180,E1 -27182.89,E2 -27182.89} C_VEL
LIN {X 0,Y 138.628,Z 228.916,A -85,B 0,C 180,E1 -27190.228,E2 -27190.228} C_VEL
LIN {X 0,Y 139.667,Z 230.116,A -85,B 0,C 180,E1 -27197.574,E2 -27197.574} C_VEL
LIN {X 0,Y 141.496,Z 233.741,A -85,B 0,C 180,E1 -27202.823,E2 -27202.823} C_VEL
LIN {X 0,Y 142.266,Z 235.041,A -85,B 0,C 180,E1 -27204.401,E2 -27204.401} C_VEL
LIN {X 0,Y 144.389,Z 238.701,A -85,B 0,C 180,E1 -27208.009,E2 -27208.009} C_VEL
LIN {X 0,Y 146.795,Z 243.272,A -85,B 0,C 180,E1 -27211.463,E2 -27211.463} C_VEL
LIN {X 0,Y 149.476,Z 248.532,A -85,B 0,C 180,E1 -27214.671,E2 -27214.671} C_VEL
LIN {X 0,Y 153.299,Z 256.525,A -85,B 0,C 180,E1 -27218.54,E2 -27218.54} C_VEL
LIN {X 0,Y 156.281,Z 263.684,A -85,B 0,C 180,E1 -27221.213,E2 -27221.213} C_VEL
LIN {X 0,Y 150.541,Z 319.872,A -85,B 0,C 180,E1 -27222.994,E2 -27222.994} C_VEL
LIN {X 0,Y 147.773,Z 335.432,A -85,B 0,C 180,E1 -27223.835,E2 -27223.835} C_VEL
LIN {X 0,Y 144.063,Z 350.092,A -85,B 0,C 180,E1 -27224.977,E2 -27224.977} C_VEL
LIN {X 0,Y 139.267,Z 364.705,A -85,B 0,C 180,E1 -27226.56,E2 -27226.56} C_VEL
LIN {X 0,Y 133.919,Z 378.04,A -85,B 0,C 180,E1 -27228.503,E2 -27228.503} C_VEL
LIN {X 0,Y 127.426,Z 391.617,A -85,B 0,C 180,E1 -27231.142,E2 -27231.142} C_VEL
LIN {X 0,Y 120.467,Z 403.985,A -85,B 0,C 180,E1 -27234.309,E2 -27234.309} C_VEL
LIN {X 0,Y 113.359,Z 415.249,A -85,B 0,C 180,E1 -27238.197,E2 -27238.197} C_VEL
LIN {X 0,Y 106.781,Z 424.734,A -85,B 0,C 180,E1 -27242.565,E2 -27242.565} C_VEL
LIN {X 0,Y 99.966,Z 434.037,A -85,B 0,C 180,E1 -27248.338,E2 -27248.338} C_VEL
LIN {X 0,Y 93.523,Z 442.686,A -85,B 0,C 180,E1 -27255.751,E2 -27255.751} C_VEL
LIN {X 0,Y 88.989,Z 448.989,A -85,B 0,C 180,E1 -27263.195,E2 -27263.195} C_VEL
LIN {X 0,Y 85.504,Z 454.684,A -85,B 0,C 180,E1 -27272.353,E2 -27272.353} C_VEL
LIN {X 0,Y 83.812,Z 458.08,A -85,B 0,C 180,E1 -27279.653,E2 -27279.653} C_VEL
LIN {X 0,Y 83.228,Z 461.45,A -85,B 0,C 180,E1 -27289.739,E2 -27289.739} C_VEL
LIN {X 0,Y 84.302,Z 463.559,A -85,B 0,C 180,E1 -27300.011,E2 -27300.011} C_VEL
LIN {X 0,Y 87.451,Z 464.384,A -85,B 0,C 180,E1 -27310.007,E2 -27310.007} C_VEL
LIN {X 0,Y 92.79,Z 463.917,A -85,B 0,C 180,E1 -27319.234,E2 -27319.234} C_VEL
LIN {X 0,Y 100.104,Z 462.134,A -85,B 0,C 180,E1 -27327.401,E2 -27327.401} C_VEL
LIN {X 0,Y 109.113,Z 458.977,A -85,B 0,C 180,E1 -27334.386,E2 -27334.386} C_VEL
LIN {X 0,Y 119.476,Z 454.364,A -85,B 0,C 180,E1 -27340.246,E2 -27340.246} C_VEL
LIN {X 0,Y 130.878,Z 448.171,A -85,B 0,C 180,E1 -27345.141,E2 -27345.141} C_VEL
LIN {X 0,Y 140.647,Z 441.887,A -85,B 0,C 180,E1 -27348.469,E2 -27348.469} C_VEL
LIN {X 0,Y 151.763,Z 433.574,A -85,B 0,C 180,E1 -27351.555,E2 -27351.555} C_VEL
LIN {X 0,Y 162.508,Z 424.126,A -85,B 0,C 180,E1 -27354.083,E2 -27354.083} C_VEL
LIN {X 0,Y 170.89,Z 415.683,A -85,B 0,C 180,E1 -27355.781,E2 -27355.781} C_VEL
LIN {X 0,Y 180.297,Z 404.716,A -85,B 0,C 180,E1 -27357.455,E2 -27357.455} C_VEL
LIN {X 0,Y 189.783,Z 391.529,A -85,B 0,C 180,E1 -27358.993,E2 -27358.993} C_VEL
LIN {X 0,Y 197.661,Z 378.387,A -85,B 0,C 180,E1 -27360.131,E2 -27360.131} C_VEL
LIN {X 0,Y 204.281,Z 364.971,A -85,B 0,C 180,E1 -27361.014,E2 -27361.014} C_VEL
LIN {X 0,Y 209.673,Z 351.321,A -85,B 0,C 180,E1 -27361.715,E2 -27361.715} C_VEL
LIN {X 0,Y 214.238,Z 336.316,A -85,B 0,C 180,E1 -27362.246,E2 -27362.246} C_VEL
LIN {X 0,Y 217.493,Z 320.997,A -85,B 0,C 180,E1 -27362.641,E2 -27362.641} C_VEL
LIN {X 0,Y 218.879,Z 311.11,A -85,B 0,C 180,E1 -27362.847,E2 -27362.847} C_VEL
LIN {X 0,Y 218.195,Z 308.738,A -85,B 0,C 180,E1 -27365.544,E2 -27365.544} C_VEL
LIN {X 0,Y 217.728,Z 308.003,A -85,B 0,C 180,E1 -27369.287,E2 -27369.287} C_VEL
LIN {X 0,Y 218.259,Z 309.216,A -85,B 0,C 180,E1 -27373.542,E2 -27373.542} C_VEL
LIN {X 0,Y 218.846,Z 311.467,A -85,B 0,C 180,E1 -27375.841,E2 -27375.841} C_VEL
LIN {X 0,Y 216.257,Z 328.259,A -85,B 0,C 180,E1 -27376.222,E2 -27376.222} C_VEL
LIN {X 0,Y 212.458,Z 343.605,A -85,B 0,C 180,E1 -27376.613,E2 -27376.613} C_VEL
LIN {X 0,Y 207.716,Z 357.601,A -85,B 0,C 180,E1 -27377.095,E2 -27377.095} C_VEL
LIN {X 0,Y 201.959,Z 370.995,A -85,B 0,C 180,E1 -27377.708,E2 -27377.708} C_VEL
LIN {X 0,Y 194.622,Z 384.86,A -85,B 0,C 180,E1 -27378.576,E2 -27378.576} C_VEL
LIN {X 0,Y 186.565,Z 397.488,A -85,B 0,C 180,E1 -27379.652,E2 -27379.652} C_VEL
LIN {X 0,Y 178.533,Z 408.19,A -85,B 0,C 180,E1 -27380.798,E2 -27380.798} C_VEL
LIN {X 0,Y 169.221,Z 418.998,A -85,B 0,C 180,E1 -27382.472,E2 -27382.472} C_VEL
LIN {X 0,Y 158.46,Z 429.615,A -85,B 0,C 180,E1 -27384.605,E2 -27384.605} C_VEL
LIN {X 0,Y 147.944,Z 438.517,A -85,B 0,C 180,E1 -27387.04,E2 -27387.04} C_VEL
LIN {X 0,Y 137.782,Z 445.925,A -85,B 0,C 180,E1 -27389.874,E2 -27389.874} C_VEL
LIN {X 0,Y 126.484,Z 453.008,A -85,B 0,C 180,E1 -27393.754,E2 -27393.754} C_VEL
LIN {X 0,Y 116.505,Z 458.422,A -85,B 0,C 180,E1 -27398.354,E2 -27398.354} C_VEL
LIN {X 0,Y 107.126,Z 462.688,A -85,B 0,C 180,E1 -27403.81,E2 -27403.81} C_VEL
LIN {X 0,Y 98.946,Z 465.78,A -85,B 0,C 180,E1 -27410.266,E2 -27410.266} C_VEL
LIN {X 0,Y 92.242,Z 467.742,A -85,B 0,C 180,E1 -27417.771,E2 -27417.771} C_VEL
LIN {X 0,Y 87.442,Z 468.568,A -85,B 0,C 180,E1 -27426.307,E2 -27426.307} C_VEL
LIN {X 0,Y 84.644,Z 468.334,A -85,B 0,C 180,E1 -27435.578,E2 -27435.578} C_VEL
LIN {X 0,Y 83.76,Z 467.014,A -85,B 0,C 180,E1 -27445.189,E2 -27445.189} C_VEL
LIN {X 0,Y 83.937,Z 465.928,A -85,B 0,C 180,E1 -27450.002,E2 -27450.002} C_VEL
LIN {X 0,Y 83.799,Z 464.482,A -85,B 0,C 180,E1 -27454.813,E2 -27454.813} C_VEL
LIN {X 0,Y 84.601,Z 460.583,A -85,B 0,C 180,E1 -27464.433,E2 -27464.433} C_VEL
LIN {X 0,Y 87.169,Z 455.293,A -85,B 0,C 180,E1 -27473.776,E2 -27473.776} C_VEL
LIN {X 0,Y 91.824,Z 448.296,A -85,B 0,C 180,E1 -27482.661,E2 -27482.661} C_VEL
LIN {X 0,Y 97.959,Z 439.954,A -85,B 0,C 180,E1 -27490.221,E2 -27490.221} C_VEL
LIN {X 0,Y 104.748,Z 430.815,A -85,B 0,C 180,E1 -27496.162,E2 -27496.162} C_VEL
LIN {X 0,Y 108.648,Z 425.222,A -85,B 0,C 180,E1 -27499.048,E2 -27499.048} C_VEL
LIN {X 0,Y 110.833,Z 421.294,A -85,B 0,C 180,E1 -27501.057,E2 -27501.057} C_VEL
LIN {X 0,Y 113.17,Z 414.579,A -85,B 0,C 180,E1 -27504.602,E2 -27504.602} C_VEL
LIN {X 0,Y 115.692,Z 407.534,A -85,B 0,C 180,E1 -27507.859,E2 -27507.859} C_VEL
LIN {X 0,Y 118.003,Z 402.984,A -85,B 0,C 180,E1 -27509.337,E2 -27509.337} C_VEL
LIN {X 0,Y 125.209,Z 390.09,A -85,B 0,C 180,E1 -27512.138,E2 -27512.138} C_VEL
LIN {X 0,Y 131.621,Z 376.581,A -85,B 0,C 180,E1 -27514.3,E2 -27514.3} C_VEL
LIN {X 0,Y 137.065,Z 362.503,A -85,B 0,C 180,E1 -27516.016,E2 -27516.016} C_VEL
LIN {X 0,Y 141.518,Z 348.442,A -85,B 0,C 180,E1 -27517.2,E2 -27517.2} C_VEL
LIN {X 0,Y 144.962,Z 333.548,A -85,B 0,C 180,E1 -27518.164,E2 -27518.164} C_VEL
LIN {X 0,Y 147.325,Z 318.996,A -85,B 0,C 180,E1 -27518.737,E2 -27518.737} C_VEL
LIN {X 0,Y 152.494,Z 268.578,A -85,B 0,C 180,E1 -27520.285,E2 -27520.285} C_VEL
LIN {X 0,Y 150.65,Z 262.04,A -85,B 0,C 180,E1 -27522.308,E2 -27522.308} C_VEL
LIN {X 0,Y 147.366,Z 254.562,A -85,B 0,C 180,E1 -27525.942,E2 -27525.942} C_VEL
LIN {X 0,Y 144.699,Z 248.943,A -85,B 0,C 180,E1 -27529.441,E2 -27529.441} C_VEL
LIN {X 0,Y 142.471,Z 244.24,A -85,B 0,C 180,E1 -27533.008,E2 -27533.008} C_VEL
LIN {X 0,Y 140.169,Z 239.916,A -85,B 0,C 180,E1 -27537.64,E2 -27537.64} C_VEL
LIN {X 0,Y 138.561,Z 236.39,A -85,B 0,C 180,E1 -27542.909,E2 -27542.909} C_VEL
LIN {X 0,Y 137.731,Z 235.97,A -85,B 0,C 180,E1 -27550.296,E2 -27550.296} C_VEL
LIN {X 0,Y 138.607,Z 237.049,A -85,B 0,C 180,E1 -27557.02,E2 -27557.02} C_VEL
LIN {X 0,Y 140.372,Z 240.682,A -85,B 0,C 180,E1 -27562.422,E2 -27562.422} C_VEL
LIN {X 0,Y 142.75,Z 245.14,A -85,B 0,C 180,E1 -27567.015,E2 -27567.015} C_VEL
LIN {X 0,Y 145.69,Z 251.019,A -85,B 0,C 180,E1 -27571.411,E2 -27571.411} C_VEL
LIN {X 0,Y 149.147,Z 258.578,A -85,B 0,C 180,E1 -27575.581,E2 -27575.581} C_VEL
LIN {X 0,Y 152,Z 265.478,A -85,B 0,C 180,E1 -27578.531,E2 -27578.531} C_VEL
LIN {X 0,Y 152.531,Z 267.131,A -85,B 0,C 180,E1 -27579.074,E2 -27579.074} C_VEL
LIN {X 0,Y 147.019,Z 319.152,A -85,B 0,C 180,E1 -27580.633,E2 -27580.633} C_VEL
LIN {X 0,Y 144.138,Z 335.055,A -85,B 0,C 180,E1 -27581.437,E2 -27581.437} C_VEL
LIN {X 0,Y 140.19,Z 350.236,A -85,B 0,C 180,E1 -27582.58,E2 -27582.58} C_VEL
LIN {X 0,Y 135.588,Z 363.945,A -85,B 0,C 180,E1 -27584.01,E2 -27584.01} C_VEL
LIN {X 0,Y 130.033,Z 377.427,A -85,B 0,C 180,E1 -27585.902,E2 -27585.902} C_VEL
LIN {X 0,Y 123.924,Z 389.887,A -85,B 0,C 180,E1 -27588.211,E2 -27588.211} C_VEL
LIN {X 0,Y 117.167,Z 401.741,A -85,B 0,C 180,E1 -27591.089,E2 -27591.089} C_VEL
LIN {X 0,Y 109.74,Z 413.195,A -85,B 0,C 180,E1 -27594.802,E2 -27594.802} C_VEL
LIN {X 0,Y 102.693,Z 423.029,A -85,B 0,C 180,E1 -27599.116,E2 -27599.116} C_VEL
LIN {X 0,Y 95.308,Z 432.651,A -85,B 0,C 180,E1 -27604.91,E2 -27604.91} C_VEL
LIN {X 0,Y 88.851,Z 440.75,A -85,B 0,C 180,E1 -27611.662,E2 -27611.662} C_VEL
LIN {X 0,Y 83.013,Z 448.144,A -85,B 0,C 180,E1 -27620.25,E2 -27620.25} C_VEL
LIN {X 0,Y 78.944,Z 454.075,A -85,B 0,C 180,E1 -27629.998,E2 -27629.998} C_VEL
LIN {X 0,Y 76.969,Z 457.633,A -85,B 0,C 180,E1 -27637.87,E2 -27637.87} C_VEL
LIN {X 0,Y 76.11,Z 460.414,A -85,B 0,C 180,E1 -27646.08,E2 -27646.08} C_VEL
LIN {X 0,Y 76.256,Z 462.137,A -85,B 0,C 180,E1 -27652.827,E2 -27652.827} C_VEL
LIN {X 0,Y 77.752,Z 463.885,A -85,B 0,C 180,E1 -27662.841,E2 -27662.841} C_VEL
LIN {X 0,Y 81.649,Z 464.617,A -85,B 0,C 180,E1 -27673.517,E2 -27673.517} C_VEL
LIN {X 0,Y 87.889,Z 464.037,A -85,B 0,C 180,E1 -27683.094,E2 -27683.094} C_VEL
LIN {X 0,Y 96.106,Z 462.123,A -85,B 0,C 180,E1 -27691.343,E2 -27691.343} C_VEL
LIN {X 0,Y 105.958,Z 458.83,A -85,B 0,C 180,E1 -27698.213,E2 -27698.213} C_VEL
LIN {X 0,Y 117.066,Z 454.075,A -85,B 0,C 180,E1 -27703.848,E2 -27703.848} C_VEL
LIN {X 0,Y 126.611,Z 449.108,A -85,B 0,C 180,E1 -27707.63,E2 -27707.63} C_VEL
LIN {X 0,Y 137.91,Z 442.213,A -85,B 0,C 180,E1 -27711.205,E2 -27711.205} C_VEL
LIN {X 0,Y 148.424,Z 434.704,A -85,B 0,C 180,E1 -27713.909,E2 -27713.909} C_VEL
LIN {X 0,Y 158.489,Z 426.365,A -85,B 0,C 180,E1 -27716.133,E2 -27716.133} C_VEL
LIN {X 0,Y 168.768,Z 416.442,A -85,B 0,C 180,E1 -27718.05,E2 -27718.05} C_VEL
LIN {X 0,Y 178.428,Z 405.484,A -85,B 0,C 180,E1 -27719.624,E2 -27719.624} C_VEL
LIN {X 0,Y 188.029,Z 392.554,A -85,B 0,C 180,E1 -27721.057,E2 -27721.057} C_VEL
LIN {X 0,Y 196.272,Z 379.17,A -85,B 0,C 180,E1 -27722.142,E2 -27722.142} C_VEL
LIN {X 0,Y 203.206,Z 365.41,A -85,B 0,C 180,E1 -27722.978,E2 -27722.978} C_VEL
LIN {X 0,Y 208.935,Z 351.115,A -85,B 0,C 180,E1 -27723.655,E2 -27723.655} C_VEL
LIN {X 0,Y 213.649,Z 335.593,A -85,B 0,C 180,E1 -27724.167,E2 -27724.167} C_VEL
LIN {X 0,Y 216.888,Z 320.146,A -85,B 0,C 180,E1 -27724.529,E2 -27724.529} C_VEL
LIN {X 0,Y 217.382,Z 316.702,A -85,B 0,C 180,E1 -27724.606,E2 -27724.606} C_VEL
LIN {X 0,Y 217.23,Z 315.782,A -85,B 0,C 180,E1 -27725.569,E2 -27725.569} C_VEL
LIN {X 0,Y 216.8,Z 315.049,A -85,B 0,C 180,E1 -27729.327,E2 -27729.327} C_VEL
LIN {X 0,Y 217.233,Z 316.167,A -85,B 0,C 180,E1 -27733.231,E2 -27733.231} C_VEL
LIN {X 0,Y 217.371,Z 317.01,A -85,B 0,C 180,E1 -27734.083,E2 -27734.083} C_VEL
LIN {X 0,Y 214.611,Z 332.118,A -85,B 0,C 180,E1 -27734.432,E2 -27734.432} C_VEL
LIN {X 0,Y 210.373,Z 347.496,A -85,B 0,C 180,E1 -27734.825,E2 -27734.825} C_VEL
LIN {X 0,Y 205.777,Z 360.177,A -85,B 0,C 180,E1 -27735.242,E2 -27735.242} C_VEL
LIN {X 0,Y 199.123,Z 374.675,A -85,B 0,C 180,E1 -27735.894,E2 -27735.894} C_VEL
LIN {X 0,Y 191.694,Z 387.839,A -85,B 0,C 180,E1 -27736.704,E2 -27736.704} C_VEL
LIN {X 0,Y 182.694,Z 401.044,A -85,B 0,C 180,E1 -27737.809,E2 -27737.809} C_VEL
LIN {X 0,Y 173.376,Z 412.572,A -85,B 0,C 180,E1 -27739.107,E2 -27739.107} C_VEL
LIN {X 0,Y 163.501,Z 423.041,A -85,B 0,C 180,E1 -27740.788,E2 -27740.788} C_VEL
LIN {X 0,Y 152.529,Z 432.939,A -85,B 0,C 180,E1 -27742.852,E2 -27742.852} C_VEL
LIN {X 0,Y 141.865,Z 441.201,A -85,B 0,C 180,E1 -27745.299,E2 -27745.299} C_VEL
LIN {X 0,Y 131.466,Z 448.143,A -85,B 0,C 180,E1 -27748.11,E2 -27748.11} C_VEL
LIN {X 0,Y 120.623,Z 454.375,A -85,B 0,C 180,E1 -27751.771,E2 -27751.771} C_VEL
LIN {X 0,Y 109.656,Z 459.758,A -85,B 0,C 180,E1 -27756.763,E2 -27756.763} C_VEL
LIN {X 0,Y 102.298,Z 462.757,A -85,B 0,C 180,E1 -27760.915,E2 -27760.915} C_VEL
LIN {X 0,Y 93.558,Z 465.748,A -85,B 0,C 180,E1 -27767.465,E2 -27767.465} C_VEL
LIN {X 0,Y 86.25,Z 467.634,A -85,B 0,C 180,E1 -27775.225,E2 -27775.225} C_VEL
LIN {X 0,Y 80.928,Z 468.391,A -85,B 0,C 180,E1 -27784.267,E2 -27784.267} C_VEL
LIN {X 0,Y 77.759,Z 468.061,A -85,B 0,C 180,E1 -27794.27,E2 -27794.27} C_VEL
LIN {X 0,Y 76.695,Z 466.647,A -85,B 0,C 180,E1 -27804.744,E2 -27804.744} C_VEL
LIN {X 0,Y 76.841,Z 465.511,A -85,B 0,C 180,E1 -27810.002,E2 -27810.002} C_VEL
LIN {X 0,Y 76.724,Z 464.03,A -85,B 0,C 180,E1 -27815.258,E2 -27815.258} C_VEL
LIN {X 0,Y 77.668,Z 460.058,A -85,B 0,C 180,E1 -27825.753,E2 -27825.753} C_VEL
LIN {X 0,Y 80.652,Z 454.661,A -85,B 0,C 180,E1 -27835.832,E2 -27835.832} C_VEL
LIN {X 0,Y 85.718,Z 447.733,A -85,B 0,C 180,E1 -27845.027,E2 -27845.027} C_VEL
LIN {X 0,Y 91.616,Z 440.214,A -85,B 0,C 180,E1 -27852.164,E2 -27852.164} C_VEL
LIN {X 0,Y 98.782,Z 431.172,A -85,B 0,C 180,E1 -27858.337,E2 -27858.337} C_VEL
LIN {X 0,Y 105.563,Z 421.889,A -85,B 0,C 180,E1 -27863.03,E2 -27863.03} C_VEL
LIN {X 0,Y 113.093,Z 410.951,A -85,B 0,C 180,E1 -27867.031,E2 -27867.031} C_VEL
LIN {X 0,Y 118.003,Z 402.984,A -85,B 0,C 180,E1 -27869.337,E2 -27869.337} C_VEL
LIN {X 0,Y 120.322,Z 398.371,A -85,B 0,C 180,E1 -27870.713,E2 -27870.713} C_VEL
LIN {X 0,Y 122.89,Z 390.605,A -85,B 0,C 180,E1 -27873.341,E2 -27873.341} C_VEL
LIN {X 0,Y 125.322,Z 382.56,A -85,B 0,C 180,E1 -27875.762,E2 -27875.762} C_VEL
LIN {X 0,Y 127.287,Z 377.436,A -85,B 0,C 180,E1 -27876.78,E2 -27876.78} C_VEL
LIN {X 0,Y 132.778,Z 363.958,A -85,B 0,C 180,E1 -27878.409,E2 -27878.409} C_VEL
LIN {X 0,Y 137.729,Z 349.033,A -85,B 0,C 180,E1 -27879.662,E2 -27879.662} C_VEL
LIN {X 0,Y 141.333,Z 334.144,A -85,B 0,C 180,E1 -27880.608,E2 -27880.608} C_VEL
LIN {X 0,Y 143.884,Z 319.188,A -85,B 0,C 180,E1 -27881.174,E2 -27881.174} C_VEL
LIN {X 0,Y 148.927,Z 270.862,A -85,B 0,C 180,E1 -27882.674,E2 -27882.674} C_VEL
LIN {X 0,Y 147.81,Z 266.82,A -85,B 0,C 180,E1 -27884.046,E2 -27884.046} C_VEL
LIN {X 0,Y 145.044,Z 260.035,A -85,B 0,C 180,E1 -27887.462,E2 -27887.462} C_VEL
LIN {X 0,Y 142.689,Z 254.746,A -85,B 0,C 180,E1 -27890.902,E2 -27890.902} C_VEL
LIN {X 0,Y 140.664,Z 250.334,A -85,B 0,C 180,E1 -27894.451,E2 -27894.451} C_VEL
LIN {X 0,Y 138.834,Z 246.536,A -85,B 0,C 180,E1 -27898.619,E2 -27898.619} C_VEL
LIN {X 0,Y 137.553,Z 243.399,A -85,B 0,C 180,E1 -27903.323,E2 -27903.323} C_VEL
LIN {X 0,Y 136.834,Z 243.027,A -85,B 0,C 180,E1 -27910.364,E2 -27910.364} C_VEL
LIN {X 0,Y 137.56,Z 243.99,A -85,B 0,C 180,E1 -27916.457,E2 -27916.457} C_VEL
LIN {X 0,Y 139.471,Z 248.229,A -85,B 0,C 180,E1 -27922.575,E2 -27922.575} C_VEL
LIN {X 0,Y 141.337,Z 252.005,A -85,B 0,C 180,E1 -27926.336,E2 -27926.336} C_VEL
LIN {X 0,Y 143.719,Z 257.045,A -85,B 0,C 180,E1 -27930.157,E2 -27930.157} C_VEL
LIN {X 0,Y 146.814,Z 264.408,A -85,B 0,C 180,E1 -27934.27,E2 -27934.27} C_VEL
LIN {X 0,Y 148.917,Z 269.833,A -85,B 0,C 180,E1 -27936.679,E2 -27936.679} C_VEL
LIN {X 0,Y 143.437,Z 320.226,A -85,B 0,C 180,E1 -27938.205,E2 -27938.205} C_VEL
LIN {X 0,Y 140.469,Z 335.928,A -85,B 0,C 180,E1 -27939.005,E2 -27939.005} C_VEL
LIN {X 0,Y 136.573,Z 350.382,A -85,B 0,C 180,E1 -27940.05,E2 -27940.05} C_VEL
LIN {X 0,Y 131.462,Z 365.012,A -85,B 0,C 180,E1 -27941.542,E2 -27941.542} C_VEL
LIN {X 0,Y 125.731,Z 378.358,A -85,B 0,C 180,E1 -27943.39,E2 -27943.39} C_VEL
LIN {X 0,Y 119.395,Z 390.701,A -85,B 0,C 180,E1 -27945.651,E2 -27945.651} C_VEL
LIN {X 0,Y 111.854,Z 403.277,A -85,B 0,C 180,E1 -27948.716,E2 -27948.716} C_VEL
LIN {X 0,Y 103.987,Z 414.72,A -85,B 0,C 180,E1 -27952.534,E2 -27952.534} C_VEL
LIN {X 0,Y 95.459,Z 425.834,A -85,B 0,C 180,E1 -27957.737,E2 -27957.737} C_VEL
LIN {X 0,Y 87.809,Z 435.024,A -85,B 0,C 180,E1 -27963.881,E2 -27963.881} C_VEL
LIN {X 0,Y 80.4,Z 443.639,A -85,B 0,C 180,E1 -27972.183,E2 -27972.183} C_VEL
LIN {X 0,Y 74.66,Z 450.567,A -85,B 0,C 180,E1 -27981.881,E2 -27981.881} C_VEL
LIN {X 0,Y 71.679,Z 454.748,A -85,B 0,C 180,E1 -27989.998,E2 -27989.998} C_VEL
LIN {X 0,Y 69.296,Z 459.179,A -85,B 0,C 180,E1 -28001.701,E2 -28001.701} C_VEL
LIN {X 0,Y 69.22,Z 462.313,A -85,B 0,C 180,E1 -28013.959,E2 -28013.959} C_VEL
LIN {X 0,Y 71.406,Z 464.196,A -85,B 0,C 180,E1 -28026.192,E2 -28026.192} C_VEL
LIN {X 0,Y 76.186,Z 464.802,A -85,B 0,C 180,E1 -28037.557,E2 -28037.557} C_VEL
LIN {X 0,Y 83.419,Z 464.108,A -85,B 0,C 180,E1 -28047.401,E2 -28047.401} C_VEL
LIN {X 0,Y 92.597,Z 462.085,A -85,B 0,C 180,E1 -28055.61,E2 -28055.61} C_VEL
LIN {X 0,Y 103.317,Z 458.666,A -85,B 0,C 180,E1 -28062.233,E2 -28062.233} C_VEL
LIN {X 0,Y 115.132,Z 453.76,A -85,B 0,C 180,E1 -28067.599,E2 -28067.599} C_VEL
LIN {X 0,Y 124.544,Z 449.02,A -85,B 0,C 180,E1 -28070.924,E2 -28070.924} C_VEL
LIN {X 0,Y 135.536,Z 442.563,A -85,B 0,C 180,E1 -28074.046,E2 -28074.046} C_VEL
LIN {X 0,Y 146.098,Z 435.298,A -85,B 0,C 180,E1 -28076.518,E2 -28076.518} C_VEL
LIN {X 0,Y 156.417,Z 427.025,A -85,B 0,C 180,E1 -28078.6,E2 -28078.6} C_VEL
LIN {X 0,Y 167.395,Z 416.7,A -85,B 0,C 180,E1 -28080.448,E2 -28080.448} C_VEL
LIN {X 0,Y 176.828,Z 406.232,A -85,B 0,C 180,E1 -28081.84,E2 -28081.84} C_VEL
LIN {X 0,Y 186.523,Z 393.525,A -85,B 0,C 180,E1 -28083.158,E2 -28083.158} C_VEL
LIN {X 0,Y 194.792,Z 380.488,A -85,B 0,C 180,E1 -28084.137,E2 -28084.137} C_VEL
LIN {X 0,Y 201.919,Z 366.779,A -85,B 0,C 180,E1 -28084.921,E2 -28084.921} C_VEL
LIN {X 0,Y 207.34,Z 353.792,A -85,B 0,C 180,E1 -28085.522,E2 -28085.522} C_VEL
LIN {X 0,Y 212.326,Z 338.444,A -85,B 0,C 180,E1 -28085.989,E2 -28085.989} C_VEL
LIN {X 0,Y 215.775,Z 323.42,A -85,B 0,C 180,E1 -28086.332,E2 -28086.332} C_VEL
LIN {X 0,Y 215.923,Z 322.573,A -85,B 0,C 180,E1 -28086.422,E2 -28086.422} C_VEL
LIN {X 0,Y 215.707,Z 322.067,A -85,B 0,C 180,E1 -28089.375,E2 -28089.375} C_VEL
LIN {X 0,Y 215.95,Z 322.768,A -85,B 0,C 180,E1 -28092.317,E2 -28092.317} C_VEL
LIN {X 0,Y 212.54,Z 338.147,A -85,B 0,C 180,E1 -28092.684,E2 -28092.684} C_VEL
LIN {X 0,Y 207.842,Z 352.992,A -85,B 0,C 180,E1 -28093.028,E2 -28093.028} C_VEL
LIN {X 0,Y 202.369,Z 366.382,A -85,B 0,C 180,E1 -28093.495,E2 -28093.495} C_VEL
LIN {X 0,Y 195.645,Z 379.589,A -85,B 0,C 180,E1 -28094.096,E2 -28094.096} C_VEL
LIN {X 0,Y 187.3,Z 393.092,A -85,B 0,C 180,E1 -28094.94,E2 -28094.94} C_VEL
LIN {X 0,Y 178.186,Z 405.373,A -85,B 0,C 180,E1 -28095.978,E2 -28095.978} C_VEL
LIN {X 0,Y 169.205,Z 415.689,A -85,B 0,C 180,E1 -28097.195,E2 -28097.195} C_VEL
LIN {X 0,Y 157.921,Z 426.772,A -85,B 0,C 180,E1 -28098.972,E2 -28098.972} C_VEL
LIN {X 0,Y 146.777,Z 436.025,A -85,B 0,C 180,E1 -28100.983,E2 -28100.983} C_VEL
LIN {X 0,Y 137.451,Z 442.775,A -85,B 0,C 180,E1 -28103.024,E2 -28103.024} C_VEL
LIN {X 0,Y 125.281,Z 450.269,A -85,B 0,C 180,E1 -28106.162,E2 -28106.162} C_VEL
LIN {X 0,Y 113.697,Z 456.276,A -85,B 0,C 180,E1 -28110.075,E2 -28110.075} C_VEL
LIN {X 0,Y 102.879,Z 460.948,A -85,B 0,C 180,E1 -28114.942,E2 -28114.942} C_VEL
LIN {X 0,Y 92.954,Z 464.412,A -85,B 0,C 180,E1 -28120.883,E2 -28120.883} C_VEL
LIN {X 0,Y 84.222,Z 466.745,A -85,B 0,C 180,E1 -28128.123,E2 -28128.123} C_VEL
LIN {X 0,Y 77.244,Z 468.001,A -85,B 0,C 180,E1 -28136.916,E2 -28136.916} C_VEL
LIN {X 0,Y 72.378,Z 468.132,A -85,B 0,C 180,E1 -28147.147,E2 -28147.147} C_VEL
LIN {X 0,Y 69.975,Z 467.171,A -85,B 0,C 180,E1 -28158.414,E2 -28158.414} C_VEL
LIN {X 0,Y 69.738,Z 465.094,A -85,B 0,C 180,E1 -28170.002,E2 -28170.002} C_VEL
LIN {X 0,Y 69.625,Z 463.561,A -85,B 0,C 180,E1 -28175.796,E2 -28175.796} C_VEL
LIN {X 0,Y 70.799,Z 459.494,A -85,B 0,C 180,E1 -28187.328,E2 -28187.328} C_VEL
LIN {X 0,Y 74.256,Z 454.006,A -85,B 0,C 180,E1 -28198.247,E2 -28198.247} C_VEL
LIN {X 0,Y 79.935,Z 446.95,A -85,B 0,C 180,E1 -28207.987,E2 -28207.987} C_VEL
LIN {X 0,Y 86.423,Z 439.335,A -85,B 0,C 180,E1 -28215.365,E2 -28215.365} C_VEL
LIN {X 0,Y 94.13,Z 430.142,A -85,B 0,C 180,E1 -28221.628,E2 -28221.628} C_VEL
LIN {X 0,Y 101.953,Z 420.034,A -85,B 0,C 180,E1 -28226.534,E2 -28226.534} C_VEL
LIN {X 0,Y 110.002,Z 408.556,A -85,B 0,C 180,E1 -28230.52,E2 -28230.52} C_VEL
LIN {X 0,Y 117.665,Z 396.128,A -85,B 0,C 180,E1 -28233.632,E2 -28233.632} C_VEL
LIN {X 0,Y 124.933,Z 382.451,A -85,B 0,C 180,E1 -28236.086,E2 -28236.086} C_VEL
LIN {X 0,Y 127.287,Z 377.436,A -85,B 0,C 180,E1 -28236.78,E2 -28236.78} C_VEL
LIN {X 0,Y 129.169,Z 372.264,A -85,B 0,C 180,E1 -28237.75,E2 -28237.75} C_VEL
LIN {X 0,Y 131.096,Z 363.719,A -85,B 0,C 180,E1 -28239.805,E2 -28239.805} C_VEL
LIN {X 0,Y 132.844,Z 354.946,A -85,B 0,C 180,E1 -28241.633,E2 -28241.633} C_VEL
LIN {X 0,Y 134.261,Z 349.428,A -85,B 0,C 180,E1 -28242.276,E2 -28242.276} C_VEL
LIN {X 0,Y 138.11,Z 334.127,A -85,B 0,C 180,E1 -28243.203,E2 -28243.203} C_VEL
LIN {X 0,Y 140.67,Z 319.738,A -85,B 0,C 180,E1 -28243.712,E2 -28243.712} C_VEL
LIN {X 0,Y 145.683,Z 273.54,A -85,B 0,C 180,E1 -28245.08,E2 -28245.08} C_VEL
LIN {X 0,Y 144.76,Z 270.703,A -85,B 0,C 180,E1 -28246.3,E2 -28246.3} C_VEL
LIN {X 0,Y 142.421,Z 264.541,A -85,B 0,C 180,E1 -28249.643,E2 -28249.643} C_VEL
LIN {X 0,Y 139.868,Z 258.373,A -85,B 0,C 180,E1 -28254.053,E2 -28254.053} C_VEL
LIN {X 0,Y 137.698,Z 253.424,A -85,B 0,C 180,E1 -28259.165,E2 -28259.165} C_VEL
LIN {X 0,Y 136.509,Z 250.392,A -85,B 0,C 180,E1 -28263.942,E2 -28263.942} C_VEL
LIN {X 0,Y 135.946,Z 249.968,A -85,B 0,C 180,E1 -28268.923,E2 -28268.923} C_VEL
LIN {X 0,Y 136.541,Z 251.029,A -85,B 0,C 180,E1 -28276.002,E2 -28276.002} C_VEL
LIN {X 0,Y 138.158,Z 254.902,A -85,B 0,C 180,E1 -28281.716,E2 -28281.716} C_VEL
LIN {X 0,Y 139.744,Z 258.393,A -85,B 0,C 180,E1 -28285.251,E2 -28285.251} C_VEL
LIN {X 0,Y 142.098,Z 263.805,A -85,B 0,C 180,E1 -28289.328,E2 -28289.328} C_VEL
LIN {X 0,Y 144.679,Z 270.538,A -85,B 0,C 180,E1 -28293.073,E2 -28293.073} C_VEL
LIN {X 0,Y 145.608,Z 273.002,A -85,B 0,C 180,E1 -28294.258,E2 -28294.258} C_VEL
LIN {X 0,Y 140.33,Z 320.155,A -85,B 0,C 180,E1 -28295.628,E2 -28295.628} C_VEL
LIN {X 0,Y 137.261,Z 336.04,A -85,B 0,C 180,E1 -28296.404,E2 -28296.404} C_VEL
LIN {X 0,Y 133.235,Z 350.529,A -85,B 0,C 180,E1 -28297.387,E2 -28297.387} C_VEL
LIN {X 0,Y 128.36,Z 364.236,A -85,B 0,C 180,E1 -28298.717,E2 -28298.717} C_VEL
LIN {X 0,Y 122.412,Z 377.74,A -85,B 0,C 180,E1 -28300.47,E2 -28300.47} C_VEL
LIN {X 0,Y 115.826,Z 390.221,A -85,B 0,C 180,E1 -28302.63,E2 -28302.63} C_VEL
LIN {X 0,Y 108.118,Z 402.695,A -85,B 0,C 180,E1 -28305.537,E2 -28305.537} C_VEL
LIN {X 0,Y 99.729,Z 414.444,A -85,B 0,C 180,E1 -28309.316,E2 -28309.316} C_VEL
LIN {X 0,Y 91.949,Z 424.137,A -85,B 0,C 180,E1 -28313.673,E2 -28313.673} C_VEL
LIN {X 0,Y 83.648,Z 433.641,A -85,B 0,C 180,E1 -28319.725,E2 -28319.725} C_VEL
LIN {X 0,Y 76.344,Z 441.575,A -85,B 0,C 180,E1 -28327.015,E2 -28327.015} C_VEL
LIN {X 0,Y 70.274,Z 448.108,A -85,B 0,C 180,E1 -28335.519,E2 -28335.519} C_VEL
LIN {X 0,Y 65.31,Z 454.136,A -85,B 0,C 180,E1 -28346.913,E2 -28346.913} C_VEL
LIN {X 0,Y 62.902,Z 457.744,A -85,B 0,C 180,E1 -28356.412,E2 -28356.412} C_VEL
LIN {X 0,Y 61.886,Z 461.396,A -85,B 0,C 180,E1 -28369.916,E2 -28369.916} C_VEL
LIN {X 0,Y 62.34,Z 462.749,A -85,B 0,C 180,E1 -28376.801,E2 -28376.801} C_VEL
LIN {X 0,Y 65.352,Z 464.507,A -85,B 0,C 180,E1 -28390.181,E2 -28390.181} C_VEL
LIN {X 0,Y 71.168,Z 464.987,A -85,B 0,C 180,E1 -28402.184,E2 -28402.184} C_VEL
LIN {X 0,Y 79.476,Z 464.163,A -85,B 0,C 180,E1 -28412.161,E2 -28412.161} C_VEL
LIN {X 0,Y 89.649,Z 462.006,A -85,B 0,C 180,E1 -28420.17,E2 -28420.17} C_VEL
LIN {X 0,Y 101.202,Z 458.462,A -85,B 0,C 180,E1 -28426.461,E2 -28426.461} C_VEL
LIN {X 0,Y 113.712,Z 453.435,A -85,B 0,C 180,E1 -28431.44,E2 -28431.44} C_VEL
LIN {X 0,Y 123.56,Z 448.623,A -85,B 0,C 180,E1 -28434.485,E2 -28434.485} C_VEL
LIN {X 0,Y 135.423,Z 441.723,A -85,B 0,C 180,E1 -28437.427,E2 -28437.427} C_VEL
LIN {X 0,Y 147.586,Z 433.276,A -85,B 0,C 180,E1 -28439.88,E2 -28439.88} C_VEL
LIN {X 0,Y 158.198,Z 424.558,A -85,B 0,C 180,E1 -28441.707,E2 -28441.707} C_VEL
LIN {X 0,Y 168.943,Z 414.212,A -85,B 0,C 180,E1 -28443.258,E2 -28443.258} C_VEL
LIN {X 0,Y 178.784,Z 403.015,A -85,B 0,C 180,E1 -28444.508,E2 -28444.508} C_VEL
LIN {X 0,Y 188.014,Z 390.511,A -85,B 0,C 180,E1 -28445.596,E2 -28445.596} C_VEL
LIN {X 0,Y 196.055,Z 377.41,A -85,B 0,C 180,E1 -28446.42,E2 -28446.42} C_VEL
LIN {X 0,Y 203.176,Z 363.12,A -85,B 0,C 180,E1 -28447.109,E2 -28447.109} C_VEL
LIN {X 0,Y 208.362,Z 350.107,A -85,B 0,C 180,E1 -28447.584,E2 -28447.584} C_VEL
LIN {X 0,Y 212.908,Z 335.157,A -85,B 0,C 180,E1 -28447.995,E2 -28447.995} C_VEL
LIN {X 0,Y 214.359,Z 329.126,A -85,B 0,C 180,E1 -28448.154,E2 -28448.154} C_VEL
LIN {X 0,Y 214.361,Z 329.283,A -85,B 0,C 180,E1 -28450.552,E2 -28450.552} C_VEL
LIN {X 0,Y 210.653,Z 343.386,A -85,B 0,C 180,E1 -28450.856,E2 -28450.856} C_VEL
LIN {X 0,Y 205.113,Z 358.936,A -85,B 0,C 180,E1 -28451.246,E2 -28451.246} C_VEL
LIN {X 0,Y 198.304,Z 373.63,A -85,B 0,C 180,E1 -28451.752,E2 -28451.752} C_VEL
LIN {X 0,Y 190.682,Z 386.897,A -85,B 0,C 180,E1 -28452.392,E2 -28452.392} C_VEL
LIN {X 0,Y 181.425,Z 400.211,A -85,B 0,C 180,E1 -28453.276,E2 -28453.276} C_VEL
LIN {X 0,Y 172.273,Z 411.241,A -85,B 0,C 180,E1 -28454.235,E2 -28454.235} C_VEL
LIN {X 0,Y 162.333,Z 421.528,A -85,B 0,C 180,E1 -28455.577,E2 -28455.577} C_VEL
LIN {X 0,Y 150.883,Z 431.606,A -85,B 0,C 180,E1 -28457.282,E2 -28457.282} C_VEL
LIN {X 0,Y 139.585,Z 440.04,A -85,B 0,C 180,E1 -28459.26,E2 -28459.26} C_VEL
LIN {X 0,Y 128.52,Z 447.105,A -85,B 0,C 180,E1 -28461.626,E2 -28461.626} C_VEL
LIN {X 0,Y 116.215,Z 453.713,A -85,B 0,C 180,E1 -28464.893,E2 -28464.893} C_VEL
LIN {X 0,Y 104.579,Z 458.944,A -85,B 0,C 180,E1 -28469.119,E2 -28469.119} C_VEL
LIN {X 0,Y 93.553,Z 462.897,A -85,B 0,C 180,E1 -28474.277,E2 -28474.277} C_VEL
LIN {X 0,Y 83.568,Z 465.685,A -85,B 0,C 180,E1 -28480.812,E2 -28480.812} C_VEL
LIN {X 0,Y 74.916,Z 467.376,A -85,B 0,C 180,E1 -28488.955,E2 -28488.955} C_VEL
LIN {X 0,Y 68.312,Z 468.008,A -85,B 0,C 180,E1 -28499.045,E2 -28499.045} C_VEL
LIN {X 0,Y 64.094,Z 467.514,A -85,B 0,C 180,E1 -28510.797,E2 -28510.797} C_VEL
LIN {X 0,Y 62.533,Z 465.909,A -85,B 0,C 180,E1 -28523.55,E2 -28523.55} C_VEL
LIN {X 0,Y 62.657,Z 464.678,A -85,B 0,C 180,E1 -28530.003,E2 -28530.003} C_VEL
LIN {X 0,Y 62.545,Z 463.092,A -85,B 0,C 180,E1 -28536.454,E2 -28536.454} C_VEL
LIN {X 0,Y 64.001,Z 458.917,A -85,B 0,C 180,E1 -28549.237,E2 -28549.237} C_VEL
LIN {X 0,Y 68.003,Z 453.313,A -85,B 0,C 180,E1 -28561.117,E2 -28561.117} C_VEL
LIN {X 0,Y 74.396,Z 446.134,A -85,B 0,C 180,E1 -28571.4,E2 -28571.4} C_VEL
LIN {X 0,Y 81.533,Z 438.412,A -85,B 0,C 180,E1 -28578.961,E2 -28578.961} C_VEL
LIN {X 0,Y 89.816,Z 429.072,A -85,B 0,C 180,E1 -28585.25,E2 -28585.25} C_VEL
LIN {X 0,Y 97.618,Z 419.515,A -85,B 0,C 180,E1 -28589.765,E2 -28589.765} C_VEL
LIN {X 0,Y 106.627,Z 407.125,A -85,B 0,C 180,E1 -28593.907,E2 -28593.907} C_VEL
LIN {X 0,Y 114.657,Z 394.443,A -85,B 0,C 180,E1 -28596.848,E2 -28596.848} C_VEL
LIN {X 0,Y 121.43,Z 381.961,A -85,B 0,C 180,E1 -28598.954,E2 -28598.954} C_VEL
LIN {X 0,Y 128.008,Z 367.315,A -85,B 0,C 180,E1 -28600.768,E2 -28600.768} C_VEL
LIN {X 0,Y 133.023,Z 353.517,A -85,B 0,C 180,E1 -28601.993,E2 -28601.993} C_VEL
LIN {X 0,Y 134.261,Z 349.428,A -85,B 0,C 180,E1 -28602.276,E2 -28602.276} C_VEL
LIN {X 0,Y 135.609,Z 343.846,A -85,B 0,C 180,E1 -28602.861,E2 -28602.861} C_VEL
LIN {X 0,Y 136.594,Z 334.728,A -85,B 0,C 180,E1 -28604.458,E2 -28604.458} C_VEL
LIN {X 0,Y 137.207,Z 325.482,A -85,B 0,C 180,E1 -28605.949,E2 -28605.949} C_VEL
LIN {X 0,Y 137.818,Z 319.697,A -85,B 0,C 180,E1 -28606.386,E2 -28606.386} C_VEL
LIN {X 0,Y 142.65,Z 276.738,A -85,B 0,C 180,E1 -28607.579,E2 -28607.579} C_VEL
LIN {X 0,Y 140.612,Z 270.787,A -85,B 0,C 180,E1 -28610.817,E2 -28610.817} C_VEL
LIN {X 0,Y 138.203,Z 264.506,A -85,B 0,C 180,E1 -28615.402,E2 -28615.402} C_VEL
LIN {X 0,Y 136.411,Z 259.997,A -85,B 0,C 180,E1 -28620.234,E2 -28620.234} C_VEL
LIN {X 0,Y 135.561,Z 257.413,A -85,B 0,C 180,E1 -28624.169,E2 -28624.169} C_VEL
LIN {X 0,Y 135.049,Z 257.007,A -85,B 0,C 180,E1 -28628.983,E2 -28628.983} C_VEL
LIN {X 0,Y 135.509,Z 257.885,A -85,B 0,C 180,E1 -28635.333,E2 -28635.333} C_VEL
LIN {X 0,Y 136.9,Z 261.636,A -85,B 0,C 180,E1 -28640.909,E2 -28640.909} C_VEL
LIN {X 0,Y 138.461,Z 265.374,A -85,B 0,C 180,E1 -28644.687,E2 -28644.687} C_VEL
LIN {X 0,Y 140.638,Z 270.924,A -85,B 0,C 180,E1 -28648.707,E2 -28648.707} C_VEL
LIN {X 0,Y 142.523,Z 276.384,A -85,B 0,C 180,E1 -28651.71,E2 -28651.71} C_VEL
LIN {X 0,Y 140.999,Z 290.751,A -85,B 0,C 180,E1 -28652.165,E2 -28652.165} C_VEL
LIN {X 0,Y 137.382,Z 320.909,A -85,B 0,C 180,E1 -28652.976,E2 -28652.976} C_VEL
LIN {X 0,Y 134.336,Z 336.168,A -85,B 0,C 180,E1 -28653.676,E2 -28653.676} C_VEL
LIN {X 0,Y 130.21,Z 350.667,A -85,B 0,C 180,E1 -28654.6,E2 -28654.6} C_VEL
LIN {X 0,Y 124.788,Z 365.318,A -85,B 0,C 180,E1 -28655.942,E2 -28655.942} C_VEL
LIN {X 0,Y 118.678,Z 378.675,A -85,B 0,C 180,E1 -28657.62,E2 -28657.62} C_VEL
LIN {X 0,Y 111.866,Z 391.035,A -85,B 0,C 180,E1 -28659.679,E2 -28659.679} C_VEL
LIN {X 0,Y 103.729,Z 403.619,A -85,B 0,C 180,E1 -28662.536,E2 -28662.536} C_VEL
LIN {X 0,Y 95.825,Z 414.165,A -85,B 0,C 180,E1 -28665.83,E2 -28665.83} C_VEL
LIN {X 0,Y 87.617,Z 423.936,A -85,B 0,C 180,E1 -28670.079,E2 -28670.079} C_VEL
LIN {X 0,Y 78.744,Z 433.509,A -85,B 0,C 180,E1 -28676.092,E2 -28676.092} C_VEL
LIN {X 0,Y 70.345,Z 441.968,A -85,B 0,C 180,E1 -28684.056,E2 -28684.056} C_VEL
LIN {X 0,Y 63.318,Z 448.916,A -85,B 0,C 180,E1 -28693.887,E2 -28693.887} C_VEL
LIN {X 0,Y 58.022,Z 454.812,A -85,B 0,C 180,E1 -28706.525,E2 -28706.525} C_VEL
LIN {X 0,Y 55.562,Z 458.361,A -85,B 0,C 180,E1 -28717.264,E2 -28717.264} C_VEL
LIN {X 0,Y 54.865,Z 461.892,A -85,B 0,C 180,E1 -28732.596,E2 -28732.596} C_VEL
LIN {X 0,Y 57.212,Z 464.164,A -85,B 0,C 180,E1 -28747.891,E2 -28747.891} C_VEL
LIN {X 0,Y 62.805,Z 465.159,A -85,B 0,C 180,E1 -28761.561,E2 -28761.561} C_VEL
LIN {X 0,Y 71.155,Z 464.861,A -85,B 0,C 180,E1 -28772.734,E2 -28772.734} C_VEL
LIN {X 0,Y 81.553,Z 463.253,A -85,B 0,C 180,E1 -28781.428,E2 -28781.428} C_VEL
LIN {X 0,Y 93.365,Z 460.288,A -85,B 0,C 180,E1 -28788.109,E2 -28788.109} C_VEL
LIN {X 0,Y 106.153,Z 455.884,A -85,B 0,C 180,E1 -28793.25,E2 -28793.25} C_VEL
LIN {X 0,Y 119.614,Z 449.929,A -85,B 0,C 180,E1 -28797.227,E2 -28797.227} C_VEL
LIN {X 0,Y 131.761,Z 443.318,A -85,B 0,C 180,E1 -28799.999,E2 -28799.999} C_VEL
LIN {X 0,Y 144.086,Z 435.249,A -85,B 0,C 180,E1 -28802.261,E2 -28802.261} C_VEL
LIN {X 0,Y 154.988,Z 426.81,A -85,B 0,C 180,E1 -28803.98,E2 -28803.98} C_VEL
LIN {X 0,Y 165.527,Z 417.232,A -85,B 0,C 180,E1 -28805.355,E2 -28805.355} C_VEL
LIN {X 0,Y 175.968,Z 406.007,A -85,B 0,C 180,E1 -28806.549,E2 -28806.549} C_VEL
LIN {X 0,Y 185.203,Z 394.199,A -85,B 0,C 180,E1 -28807.533,E2 -28807.533} C_VEL
LIN {X 0,Y 193.935,Z 380.821,A -85,B 0,C 180,E1 -28808.334,E2 -28808.334} C_VEL
LIN {X 0,Y 200.985,Z 367.601,A -85,B 0,C 180,E1 -28808.948,E2 -28808.948} C_VEL
LIN {X 0,Y 204.307,Z 360.286,A -85,B 0,C 180,E1 -28809.244,E2 -28809.244} C_VEL
LIN {X 0,Y 197.858,Z 373.892,A -85,B 0,C 180,E1 -28809.708,E2 -28809.708} C_VEL
LIN {X 0,Y 190.161,Z 387.092,A -85,B 0,C 180,E1 -28810.263,E2 -28810.263} C_VEL
LIN {X 0,Y 180.796,Z 400.328,A -85,B 0,C 180,E1 -28811.033,E2 -28811.033} C_VEL
LIN {X 0,Y 170.829,Z 412.104,A -85,B 0,C 180,E1 -28811.937,E2 -28811.937} C_VEL
LIN {X 0,Y 160.589,Z 422.372,A -85,B 0,C 180,E1 -28813.161,E2 -28813.161} C_VEL
LIN {X 0,Y 148.942,Z 432.277,A -85,B 0,C 180,E1 -28814.692,E2 -28814.692} C_VEL
LIN {X 0,Y 137.409,Z 440.562,A -85,B 0,C 180,E1 -28816.468,E2 -28816.468} C_VEL
LIN {X 0,Y 126.08,Z 447.49,A -85,B 0,C 180,E1 -28818.63,E2 -28818.63} C_VEL
LIN {X 0,Y 113.407,Z 453.974,A -85,B 0,C 180,E1 -28821.635,E2 -28821.635} C_VEL
LIN {X 0,Y 101.285,Z 459.092,A -85,B 0,C 180,E1 -28825.575,E2 -28825.575} C_VEL
LIN {X 0,Y 89.722,Z 462.984,A -85,B 0,C 180,E1 -28830.502,E2 -28830.502} C_VEL
LIN {X 0,Y 79.083,Z 465.661,A -85,B 0,C 180,E1 -28836.89,E2 -28836.89} C_VEL
LIN {X 0,Y 69.661,Z 467.247,A -85,B 0,C 180,E1 -28845.075,E2 -28845.075} C_VEL
LIN {X 0,Y 62.287,Z 467.782,A -85,B 0,C 180,E1 -28855.659,E2 -28855.659} C_VEL
LIN {X 0,Y 57.393,Z 467.24,A -85,B 0,C 180,E1 -28868.45,E2 -28868.45} C_VEL
LIN {X 0,Y 55.483,Z 465.541,A -85,B 0,C 180,E1 -28882.726,E2 -28882.726} C_VEL
LIN {X 0,Y 55.565,Z 464.261,A -85,B 0,C 180,E1 -28890.003,E2 -28890.003} C_VEL
LIN {X 0,Y 56.036,Z 460.655,A -85,B 0,C 180,E1 -28904.53,E2 -28904.53} C_VEL
LIN {X 0,Y 59.262,Z 455.667,A -85,B 0,C 180,E1 -28918.322,E2 -28918.322} C_VEL
LIN {X 0,Y 65.263,Z 449.177,A -85,B 0,C 180,E1 -28930.253,E2 -28930.253} C_VEL
LIN {X 0,Y 72.346,Z 442.144,A -85,B 0,C 180,E1 -28938.843,E2 -28938.843} C_VEL
LIN {X 0,Y 80.728,Z 433.637,A -85,B 0,C 180,E1 -28945.8,E2 -28945.8} C_VEL
LIN {X 0,Y 89.567,Z 423.768,A -85,B 0,C 180,E1 -28951.326,E2 -28951.326} C_VEL
LIN {X 0,Y 98.506,Z 412.759,A -85,B 0,C 180,E1 -28955.463,E2 -28955.463} C_VEL
LIN {X 0,Y 106.647,Z 401.231,A -85,B 0,C 180,E1 -28958.569,E2 -28958.569} C_VEL
LIN {X 0,Y 114.339,Z 388.713,A -85,B 0,C 180,E1 -28960.922,E2 -28960.922} C_VEL
LIN {X 0,Y 121.358,Z 375.071,A -85,B 0,C 180,E1 -28962.802,E2 -28962.802} C_VEL
LIN {X 0,Y 127.421,Z 360.593,A -85,B 0,C 180,E1 -28964.258,E2 -28964.258} C_VEL
LIN {X 0,Y 132.185,Z 346.267,A -85,B 0,C 180,E1 -28965.243,E2 -28965.243} C_VEL
LIN {X 0,Y 136.011,Z 330.45,A -85,B 0,C 180,E1 -28966.047,E2 -28966.047} C_VEL
LIN {X 0,Y 137.818,Z 319.697,A -85,B 0,C 180,E1 -28966.386,E2 -28966.386} C_VEL
LIN {X 0,Y 138.317,Z 313.894,A -85,B 0,C 180,E1 -28966.807,E2 -28966.807} C_VEL
LIN {X 0,Y 138.36,Z 295.19,A -85,B 0,C 180,E1 -28969.578,E2 -28969.578} C_VEL
LIN {X 0,Y 138.823,Z 289.373,A -85,B 0,C 180,E1 -28969.949,E2 -28969.949} C_VEL
LIN {X 0,Y 139.858,Z 280.214,A -85,B 0,C 180,E1 -28970.186,E2 -28970.186} C_VEL
LIN {X 0,Y 137.796,Z 274.007,A -85,B 0,C 180,E1 -28974.066,E2 -28974.066} C_VEL
LIN {X 0,Y 136.365,Z 269.938,A -85,B 0,C 180,E1 -28977.442,E2 -28977.442} C_VEL
LIN {X 0,Y 135.235,Z 266.714,A -85,B 0,C 180,E1 -28981.088,E2 -28981.088} C_VEL
LIN {X 0,Y 134.58,Z 264.385,A -85,B 0,C 180,E1 -28984.601,E2 -28984.601} C_VEL
LIN {X 0,Y 134.142,Z 264.144,A -85,B 0,C 180,E1 -28989.924,E2 -28989.924} C_VEL
LIN {X 0,Y 134.525,Z 264.9,A -85,B 0,C 180,E1 -28994.91,E2 -28994.91} C_VEL
LIN {X 0,Y 135.698,Z 268.429,A -85,B 0,C 180,E1 -29000.175,E2 -29000.175} C_VEL
LIN {X 0,Y 137.095,Z 272.184,A -85,B 0,C 180,E1 -29003.913,E2 -29003.913} C_VEL
LIN {X 0,Y 138.845,Z 277.209,A -85,B 0,C 180,E1 -29007.497,E2 -29007.497} C_VEL
LIN {X 0,Y 139.741,Z 279.959,A -85,B 0,C 180,E1 -29009.097,E2 -29009.097} C_VEL
LIN {X 0,Y 139.163,Z 285.542,A -85,B 0,C 180,E1 -29009.308,E2 -29009.308} C_VEL
LIN {X 0,Y 134.807,Z 321.285,A -85,B 0,C 180,E1 -29010.201,E2 -29010.201} C_VEL
LIN {X 0,Y 131.749,Z 336.213,A -85,B 0,C 180,E1 -29010.828,E2 -29010.828} C_VEL
LIN {X 0,Y 127.504,Z 350.807,A -85,B 0,C 180,E1 -29011.686,E2 -29011.686} C_VEL
LIN {X 0,Y 122.352,Z 364.526,A -85,B 0,C 180,E1 -29012.849,E2 -29012.849} C_VEL
LIN {X 0,Y 116.037,Z 378.048,A -85,B 0,C 180,E1 -29014.386,E2 -29014.386} C_VEL
LIN {X 0,Y 108.983,Z 390.555,A -85,B 0,C 180,E1 -29016.282,E2 -29016.282} C_VEL
LIN {X 0,Y 100.765,Z 402.944,A -85,B 0,C 180,E1 -29018.884,E2 -29018.884} C_VEL
LIN {X 0,Y 92.302,Z 413.887,A -85,B 0,C 180,E1 -29022.063,E2 -29022.063} C_VEL
LIN {X 0,Y 83.658,Z 423.736,A -85,B 0,C 180,E1 -29026.123,E2 -29026.123} C_VEL
LIN {X 0,Y 74.188,Z 433.379,A -85,B 0,C 180,E1 -29031.99,E2 -29031.99} C_VEL
LIN {X 0,Y 65.603,Z 441.394,A -85,B 0,C 180,E1 -29039.393,E2 -29039.393} C_VEL
LIN {X 0,Y 58.237,Z 448.071,A -85,B 0,C 180,E1 -29048.772,E2 -29048.772} C_VEL
LIN {X 0,Y 51.932,Z 454.2,A -85,B 0,C 180,E1 -29062.219,E2 -29062.219} C_VEL
LIN {X 0,Y 49.239,Z 457.367,A -85,B 0,C 180,E1 -29072.303,E2 -29072.303} C_VEL
LIN {X 0,Y 47.622,Z 460.829,A -85,B 0,C 180,E1 -29087.164,E2 -29087.164} C_VEL
LIN {X 0,Y 48.31,Z 462.824,A -85,B 0,C 180,E1 -29099.2,E2 -29099.2} C_VEL
LIN {X 0,Y 51.347,Z 464.539,A -85,B 0,C 180,E1 -29113.181,E2 -29113.181} C_VEL
LIN {X 0,Y 58.282,Z 465.408,A -85,B 0,C 180,E1 -29127.571,E2 -29127.571} C_VEL
LIN {X 0,Y 67.936,Z 464.987,A -85,B 0,C 180,E1 -29138.594,E2 -29138.594} C_VEL
LIN {X 0,Y 79.406,Z 463.257,A -85,B 0,C 180,E1 -29146.793,E2 -29146.793} C_VEL
LIN {X 0,Y 92.074,Z 460.164,A -85,B 0,C 180,E1 -29152.868,E2 -29152.868} C_VEL
LIN {X 0,Y 105.522,Z 455.629,A -85,B 0,C 180,E1 -29157.447,E2 -29157.447} C_VEL
LIN {X 0,Y 119.49,Z 449.536,A -85,B 0,C 180,E1 -29160.943,E2 -29160.943} C_VEL
LIN {X 0,Y 130.434,Z 443.691,A -85,B 0,C 180,E1 -29163.087,E2 -29163.087} C_VEL
LIN {X 0,Y 143.485,Z 435.33,A -85,B 0,C 180,E1 -29165.168,E2 -29165.168} C_VEL
LIN {X 0,Y 155.711,Z 425.907,A -85,B 0,C 180,E1 -29166.806,E2 -29166.806} C_VEL
LIN {X 0,Y 167.51,Z 415.022,A -85,B 0,C 180,E1 -29168.094,E2 -29168.094} C_VEL
LIN {X 0,Y 174.271,Z 407.804,A -85,B 0,C 180,E1 -29168.745,E2 -29168.745} C_VEL
LIN {X 0,Y 173.572,Z 408.615,A -85,B 0,C 180,E1 -29169.285,E2 -29169.285} C_VEL
LIN {X 0,Y 164.216,Z 418.416,A -85,B 0,C 180,E1 -29170.158,E2 -29170.158} C_VEL
LIN {X 0,Y 152.362,Z 428.943,A -85,B 0,C 180,E1 -29171.424,E2 -29171.424} C_VEL
LIN {X 0,Y 140.593,Z 437.767,A -85,B 0,C 180,E1 -29172.901,E2 -29172.901} C_VEL
LIN {X 0,Y 127.301,Z 446.079,A -85,B 0,C 180,E1 -29174.958,E2 -29174.958} C_VEL
LIN {X 0,Y 114.206,Z 452.818,A -85,B 0,C 180,E1 -29177.481,E2 -29177.481} C_VEL
LIN {X 0,Y 104.626,Z 456.896,A -85,B 0,C 180,E1 -29179.883,E2 -29179.883} C_VEL
LIN {X 0,Y 92.302,Z 461.279,A -85,B 0,C 180,E1 -29183.982,E2 -29183.982} C_VEL
LIN {X 0,Y 80.552,Z 464.489,A -85,B 0,C 180,E1 -29189.255,E2 -29189.255} C_VEL
LIN {X 0,Y 69.754,Z 466.517,A -85,B 0,C 180,E1 -29196.293,E2 -29196.293} C_VEL
LIN {X 0,Y 60.394,Z 467.471,A -85,B 0,C 180,E1 -29205.72,E2 -29205.72} C_VEL
LIN {X 0,Y 53.246,Z 467.378,A -85,B 0,C 180,E1 -29218.135,E2 -29218.135} C_VEL
LIN {X 0,Y 49.198,Z 466.208,A -85,B 0,C 180,E1 -29233.403,E2 -29233.403} C_VEL
LIN {X 0,Y 48.461,Z 463.845,A -85,B 0,C 180,E1 -29250.003,E2 -29250.003} C_VEL
LIN {X 0,Y 49.16,Z 460.134,A -85,B 0,C 180,E1 -29266.617,E2 -29266.617} C_VEL
LIN {X 0,Y 53.064,Z 455.035,A -85,B 0,C 180,E1 -29281.994,E2 -29281.994} C_VEL
LIN {X 0,Y 59.954,Z 448.425,A -85,B 0,C 180,E1 -29294.699,E2 -29294.699} C_VEL
LIN {X 0,Y 67.815,Z 441.26,A -85,B 0,C 180,E1 -29303.438,E2 -29303.438} C_VEL
LIN {X 0,Y 76.902,Z 432.608,A -85,B 0,C 180,E1 -29310.254,E2 -29310.254} C_VEL
LIN {X 0,Y 86.553,Z 422.291,A -85,B 0,C 180,E1 -29315.677,E2 -29315.677} C_VEL
LIN {X 0,Y 95.74,Z 411.37,A -85,B 0,C 180,E1 -29319.386,E2 -29319.386} C_VEL
LIN {X 0,Y 104.224,Z 399.606,A -85,B 0,C 180,E1 -29322.27,E2 -29322.27} C_VEL
LIN {X 0,Y 112.185,Z 386.805,A -85,B 0,C 180,E1 -29324.412,E2 -29324.412} C_VEL
LIN {X 0,Y 119.003,Z 373.659,A -85,B 0,C 180,E1 -29326.036,E2 -29326.036} C_VEL
LIN {X 0,Y 125.164,Z 359.053,A -85,B 0,C 180,E1 -29327.327,E2 -29327.327} C_VEL
LIN {X 0,Y 130.046,Z 344.276,A -85,B 0,C 180,E1 -29328.226,E2 -29328.226} C_VEL
LIN {X 0,Y 133.632,Z 329.36,A -85,B 0,C 180,E1 -29328.886,E2 -29328.886} C_VEL
LIN {X 0,Y 135.884,Z 314.985,A -85,B 0,C 180,E1 -29329.332,E2 -29329.332} C_VEL
LIN {X 0,Y 138.823,Z 289.373,A -85,B 0,C 180,E1 -29329.949,E2 -29329.949} C_VEL
LIN {X 0,Y 138.885,Z 286.77,A -85,B 0,C 180,E1 -29330.304,E2 -29330.304} C_VEL
LIN {X 0,Y 138.466,Z 284.211,A -85,B 0,C 180,E1 -29331.272,E2 -29331.272} C_VEL
LIN {X 0,Y 137.686,Z 282.221,A -85,B 0,C 180,E1 -29332.653,E2 -29332.653} C_VEL
LIN {X 0,Y 135.637,Z 278.434,A -85,B 0,C 180,E1 -29336.713,E2 -29336.713} C_VEL
LIN {X 0,Y 135.435,Z 277.74,A -85,B 0,C 180,E1 -29337.274,E2 -29337.274} C_VEL
LIN {X 0,Y 134.07,Z 273.371,A -85,B 0,C 180,E1 -29342.041,E2 -29342.041} C_VEL
LIN {X 0,Y 133.574,Z 271.371,A -85,B 0,C 180,E1 -29345.219,E2 -29345.219} C_VEL
LIN {X 0,Y 133.245,Z 271.199,A -85,B 0,C 180,E1 -29349.992,E2 -29349.992} C_VEL
LIN {X 0,Y 133.53,Z 271.837,A -85,B 0,C 180,E1 -29354.32,E2 -29354.32} C_VEL
LIN {X 0,Y 134.466,Z 275.082,A -85,B 0,C 180,E1 -29359.24,E2 -29359.24} C_VEL
LIN {X 0,Y 135.626,Z 278.579,A -85,B 0,C 180,E1 -29362.784,E2 -29362.784} C_VEL
LIN {X 0,Y 137.187,Z 283.676,A -85,B 0,C 180,E1 -29366.406,E2 -29366.406} C_VEL
LIN {X 0,Y 132.57,Z 321.286,A -85,B 0,C 180,E1 -29367.317,E2 -29367.317} C_VEL
LIN {X 0,Y 129.299,Z 336.806,A -85,B 0,C 180,E1 -29367.908,E2 -29367.908} C_VEL
LIN {X 0,Y 124.736,Z 351.937,A -85,B 0,C 180,E1 -29368.733,E2 -29368.733} C_VEL
LIN {X 0,Y 119.455,Z 365.508,A -85,B 0,C 180,E1 -29369.793,E2 -29369.793} C_VEL
LIN {X 0,Y 112.966,Z 378.918,A -85,B 0,C 180,E1 -29371.189,E2 -29371.189} C_VEL
LIN {X 0,Y 105.716,Z 391.31,A -85,B 0,C 180,E1 -29372.93,E2 -29372.93} C_VEL
LIN {X 0,Y 97.148,Z 403.722,A -85,B 0,C 180,E1 -29375.365,E2 -29375.365} C_VEL
LIN {X 0,Y 87.668,Z 415.383,A -85,B 0,C 180,E1 -29378.588,E2 -29378.588} C_VEL
LIN {X 0,Y 77.175,Z 426.528,A -85,B 0,C 180,E1 -29383.234,E2 -29383.234} C_VEL
LIN {X 0,Y 67.299,Z 435.737,A -85,B 0,C 180,E1 -29389.253,E2 -29389.253} C_VEL
LIN {X 0,Y 58.071,Z 443.6,A -85,B 0,C 180,E1 -29397.461,E2 -29397.461} C_VEL
LIN {X 0,Y 49.609,Z 450.525,A -85,B 0,C 180,E1 -29409.254,E2 -29409.254} C_VEL
LIN {X 0,Y 44.724,Z 454.866,A -85,B 0,C 180,E1 -29420.955,E2 -29420.955} C_VEL
LIN {X 0,Y 42.177,Z 457.569,A -85,B 0,C 180,E1 -29430.962,E2 -29430.962} C_VEL
LIN {X 0,Y 40.529,Z 461.311,A -85,B 0,C 180,E1 -29450.289,E2 -29450.289} C_VEL
LIN {X 0,Y 41.506,Z 462.988,A -85,B 0,C 180,E1 -29462.146,E2 -29462.146} C_VEL
LIN {X 0,Y 46.02,Z 464.877,A -85,B 0,C 180,E1 -29479.776,E2 -29479.776} C_VEL
LIN {X 0,Y 54.515,Z 465.652,A -85,B 0,C 180,E1 -29494.474,E2 -29494.474} C_VEL
LIN {X 0,Y 65.484,Z 465.115,A -85,B 0,C 180,E1 -29504.991,E2 -29504.991} C_VEL
LIN {X 0,Y 77.99,Z 463.261,A -85,B 0,C 180,E1 -29512.401,E2 -29512.401} C_VEL
LIN {X 0,Y 91.433,Z 460.041,A -85,B 0,C 180,E1 -29517.728,E2 -29517.728} C_VEL
LIN {X 0,Y 105.464,Z 455.374,A -85,B 0,C 180,E1 -29521.692,E2 -29521.692} C_VEL
LIN {X 0,Y 116.525,Z 450.707,A -85,B 0,C 180,E1 -29524.042,E2 -29524.042} C_VEL
LIN {X 0,Y 129.51,Z 444.056,A -85,B 0,C 180,E1 -29526.229,E2 -29526.229} C_VEL
LIN {X 0,Y 141.91,Z 436.358,A -85,B 0,C 180,E1 -29527.917,E2 -29527.917} C_VEL
LIN {X 0,Y 149.343,Z 430.997,A -85,B 0,C 180,E1 -29528.798,E2 -29528.798} C_VEL
LIN {X 0,Y 149.401,Z 430.958,A -85,B 0,C 180,E1 -29528.942,E2 -29528.942} C_VEL
LIN {X 0,Y 137.477,Z 439.396,A -85,B 0,C 180,E1 -29530.24,E2 -29530.24} C_VEL
LIN {X 0,Y 125.66,Z 446.463,A -85,B 0,C 180,E1 -29531.837,E2 -29531.837} C_VEL
LIN {X 0,Y 112.273,Z 453.08,A -85,B 0,C 180,E1 -29534.014,E2 -29534.014} C_VEL
LIN {X 0,Y 99.189,Z 458.319,A -85,B 0,C 180,E1 -29536.959,E2 -29536.959} C_VEL
LIN {X 0,Y 89.64,Z 461.369,A -85,B 0,C 180,E1 -29539.812,E2 -29539.812} C_VEL
LIN {X 0,Y 77.315,Z 464.475,A -85,B 0,C 180,E1 -29544.635,E2 -29544.635} C_VEL
LIN {X 0,Y 65.765,Z 466.447,A -85,B 0,C 180,E1 -29551.254,E2 -29551.254} C_VEL
LIN {X 0,Y 55.495,Z 467.296,A -85,B 0,C 180,E1 -29560.554,E2 -29560.554} C_VEL
LIN {X 0,Y 47.327,Z 467.099,A -85,B 0,C 180,E1 -29573.563,E2 -29573.563} C_VEL
LIN {X 0,Y 42.421,Z 465.847,A -85,B 0,C 180,E1 -29590.653,E2 -29590.653} C_VEL
LIN {X 0,Y 41.345,Z 463.427,A -85,B 0,C 180,E1 -29610.004,E2 -29610.004} C_VEL
LIN {X 0,Y 42.351,Z 459.612,A -85,B 0,C 180,E1 -29629.388,E2 -29629.388} C_VEL
LIN {X 0,Y 47.14,Z 454.403,A -85,B 0,C 180,E1 -29646.614,E2 -29646.614} C_VEL
LIN {X 0,Y 55.077,Z 447.674,A -85,B 0,C 180,E1 -29659.967,E2 -29659.967} C_VEL
LIN {X 0,Y 63.783,Z 440.378,A -85,B 0,C 180,E1 -29668.648,E2 -29668.648} C_VEL
LIN {X 0,Y 73.587,Z 431.577,A -85,B 0,C 180,E1 -29675.142,E2 -29675.142} C_VEL
LIN {X 0,Y 83.411,Z 421.547,A -85,B 0,C 180,E1 -29680.003,E2 -29680.003} C_VEL
LIN {X 0,Y 92.649,Z 410.958,A -85,B 0,C 180,E1 -29683.279,E2 -29683.279} C_VEL
LIN {X 0,Y 101.444,Z 399.141,A -85,B 0,C 180,E1 -29685.918,E2 -29685.918} C_VEL
LIN {X 0,Y 109.64,Z 386.279,A -85,B 0,C 180,E1 -29687.839,E2 -29687.839} C_VEL
LIN {X 0,Y 116.397,Z 373.57,A -85,B 0,C 180,E1 -29689.245,E2 -29689.245} C_VEL
LIN {X 0,Y 122.526,Z 359.471,A -85,B 0,C 180,E1 -29690.363,E2 -29690.363} C_VEL
LIN {X 0,Y 127.577,Z 344.627,A -85,B 0,C 180,E1 -29691.18,E2 -29691.18} C_VEL
LIN {X 0,Y 131.346,Z 329.336,A -85,B 0,C 180,E1 -29691.793,E2 -29691.793} C_VEL
LIN {X 0,Y 133.639,Z 315.117,A -85,B 0,C 180,E1 -29692.185,E2 -29692.185} C_VEL
LIN {X 0,Y 137.287,Z 283.882,A -85,B 0,C 180,E1 -29692.903,E2 -29692.903} C_VEL
LIN {X 0,Y 135.62,Z 278.337,A -85,B 0,C 180,E1 -29696.768,E2 -29696.768} C_VEL
LIN {X 0,Y 135.435,Z 277.74,A -85,B 0,C 180,E1 -29697.274,E2 -29697.274} C_VEL
LIN {X 0,Y 134.907,Z 276.28,A -85,B 0,C 180,E1 -29698.794,E2 -29698.794} C_VEL
LIN {X 0,Y 134.063,Z 275.511,A -85,B 0,C 180,E1 -29701.265,E2 -29701.265} C_VEL
LIN {X 0,Y 133.312,Z 275.909,A -85,B 0,C 180,E1 -29703.803,E2 -29703.803} C_VEL
LIN {X 0,Y 132.393,Z 277.964,A -85,B 0,C 180,E1 -29709.113,E2 -29709.113} C_VEL
LIN {X 0,Y 132.351,Z 278.341,A -85,B 0,C 180,E1 -29710.908,E2 -29710.908} C_VEL
LIN {X 0,Y 132.561,Z 278.864,A -85,B 0,C 180,E1 -29713.879,E2 -29713.879} C_VEL
LIN {X 0,Y 133.344,Z 281.947,A -85,B 0,C 180,E1 -29718.587,E2 -29718.587} C_VEL
LIN {X 0,Y 134.287,Z 285.366,A -85,B 0,C 180,E1 -29721.896,E2 -29721.896} C_VEL
LIN {X 0,Y 134.915,Z 287.594,A -85,B 0,C 180,E1 -29723.634,E2 -29723.634} C_VEL
LIN {X 0,Y 130.691,Z 321.133,A -85,B 0,C 180,E1 -29724.347,E2 -29724.347} C_VEL
LIN {X 0,Y 127.32,Z 336.867,A -85,B 0,C 180,E1 -29724.866,E2 -29724.866} C_VEL
LIN {X 0,Y 122.724,Z 351.871,A -85,B 0,C 180,E1 -29725.581,E2 -29725.581} C_VEL
LIN {X 0,Y 116.911,Z 366.383,A -85,B 0,C 180,E1 -29726.591,E2 -29726.591} C_VEL
LIN {X 0,Y 110.266,Z 379.685,A -85,B 0,C 180,E1 -29727.825,E2 -29727.825} C_VEL
LIN {X 0,Y 102.025,Z 393.225,A -85,B 0,C 180,E1 -29729.576,E2 -29729.576} C_VEL
LIN {X 0,Y 94.002,Z 404.335,A -85,B 0,C 180,E1 -29731.559,E2 -29731.559} C_VEL
LIN {X 0,Y 84.988,Z 415.021,A -85,B 0,C 180,E1 -29734.211,E2 -29734.211} C_VEL
LIN {X 0,Y 75.546,Z 424.753,A -85,B 0,C 180,E1 -29737.741,E2 -29737.741} C_VEL
LIN {X 0,Y 64.969,Z 434.293,A -85,B 0,C 180,E1 -29743.095,E2 -29743.095} C_VEL
LIN {X 0,Y 55.077,Z 442.224,A -85,B 0,C 180,E1 -29750.352,E2 -29750.352} C_VEL
LIN {X 0,Y 45.103,Z 449.638,A -85,B 0,C 180,E1 -29762.126,E2 -29762.126} C_VEL
LIN {X 0,Y 37.527,Z 455.513,A -85,B 0,C 180,E1 -29779.202,E2 -29779.202} C_VEL
LIN {X 0,Y 34.107,Z 459.057,A -85,B 0,C 180,E1 -29795.909,E2 -29795.909} C_VEL
LIN {X 0,Y 33.573,Z 461.788,A -85,B 0,C 180,E1 -29814.746,E2 -29814.746} C_VEL
LIN {X 0,Y 34.974,Z 463.234,A -85,B 0,C 180,E1 -29827.069,E2 -29827.069} C_VEL
LIN {X 0,Y 41.469,Z 465.183,A -85,B 0,C 180,E1 -29847.921,E2 -29847.921} C_VEL
LIN {X 0,Y 51.641,Z 465.849,A -85,B 0,C 180,E1 -29862.291,E2 -29862.291} C_VEL
LIN {X 0,Y 63.907,Z 465.22,A -85,B 0,C 180,E1 -29871.772,E2 -29871.772} C_VEL
LIN {X 0,Y 77.345,Z 463.261,A -85,B 0,C 180,E1 -29878.171,E2 -29878.171} C_VEL
LIN {X 0,Y 91.459,Z 459.918,A -85,B 0,C 180,E1 -29882.64,E2 -29882.64} C_VEL
LIN {X 0,Y 105.978,Z 455.118,A -85,B 0,C 180,E1 -29885.896,E2 -29885.896} C_VEL
LIN {X 0,Y 120.741,Z 448.733,A -85,B 0,C 180,E1 -29888.309,E2 -29888.309} C_VEL
LIN {X 0,Y 120.978,Z 448.645,A -85,B 0,C 180,E1 -29889.045,E2 -29889.045} C_VEL
LIN {X 0,Y 107.387,Z 454.759,A -85,B 0,C 180,E1 -29890.991,E2 -29890.991} C_VEL
LIN {X 0,Y 94.035,Z 459.532,A -85,B 0,C 180,E1 -29893.695,E2 -29893.695} C_VEL
LIN {X 0,Y 80.975,Z 463.1,A -85,B 0,C 180,E1 -29897.314,E2 -29897.314} C_VEL
LIN {X 0,Y 68.395,Z 465.541,A -85,B 0,C 180,E1 -29902.367,E2 -29902.367} C_VEL
LIN {X 0,Y 54.934,Z 466.965,A -85,B 0,C 180,E1 -29910.776,E2 -29910.776} C_VEL
LIN {X 0,Y 46.169,Z 467.102,A -85,B 0,C 180,E1 -29920.443,E2 -29920.443} C_VEL
LIN {X 0,Y 38.275,Z 466.277,A -85,B 0,C 180,E1 -29936.579,E2 -29936.579} C_VEL
LIN {X 0,Y 34.415,Z 464.372,A -85,B 0,C 180,E1 -29958.221,E2 -29958.221} C_VEL
LIN {X 0,Y 34.248,Z 462.982,A -85,B 0,C 180,E1 -29970.005,E2 -29970.005} C_VEL
LIN {X 0,Y 35.688,Z 459.067,A -85,B 0,C 180,E1 -29993.2,E2 -29993.2} C_VEL
LIN {X 0,Y 41.587,Z 453.737,A -85,B 0,C 180,E1 -30012.536,E2 -30012.536} C_VEL
LIN {X 0,Y 51.342,Z 446.465,A -85,B 0,C 180,E1 -30026.805,E2 -30026.805} C_VEL
LIN {X 0,Y 61.82,Z 438.305,A -85,B 0,C 180,E1 -30035.439,E2 -30035.439} C_VEL
LIN {X 0,Y 72.395,Z 429.093,A -85,B 0,C 180,E1 -30041.183,E2 -30041.183} C_VEL
LIN {X 0,Y 82.96,Z 418.538,A -85,B 0,C 180,E1 -30045.279,E2 -30045.279} C_VEL
LIN {X 0,Y 92.475,Z 407.47,A -85,B 0,C 180,E1 -30048.102,E2 -30048.102} C_VEL
LIN {X 0,Y 101.622,Z 395.021,A -85,B 0,C 180,E1 -30050.243,E2 -30050.243} C_VEL
LIN {X 0,Y 110.043,Z 381.295,A -85,B 0,C 180,E1 -30051.869,E2 -30051.869} C_VEL
LIN {X 0,Y 117.036,Z 367.341,A -85,B 0,C 180,E1 -30053.033,E2 -30053.033} C_VEL
LIN {X 0,Y 122.817,Z 352.918,A -85,B 0,C 180,E1 -30053.868,E2 -30053.868} C_VEL
LIN {X 0,Y 127.482,Z 337.472,A -85,B 0,C 180,E1 -30054.542,E2 -30054.542} C_VEL
LIN {X 0,Y 130.701,Z 322.281,A -85,B 0,C 180,E1 -30054.935,E2 -30054.935} C_VEL
LIN {X 0,Y 134.957,Z 287.677,A -85,B 0,C 180,E1 -30055.759,E2 -30055.759} C_VEL
LIN {X 0,Y 133.778,Z 283.153,A -85,B 0,C 180,E1 -30059.345,E2 -30059.345} C_VEL
LIN {X 0,Y 132.939,Z 280.019,A -85,B 0,C 180,E1 -30063.032,E2 -30063.032} C_VEL
LIN {X 0,Y 132.606,Z 278.387,A -85,B 0,C 180,E1 -30065.671,E2 -30065.671} C_VEL
LIN {X 0,Y 132.348,Z 278.256,A -85,B 0,C 180,E1 -30070.06,E2 -30070.06} C_VEL
LIN {X 0,Y 132.351,Z 278.341,A -85,B 0,C 180,E1 -30070.908,E2 -30070.908} C_VEL
LIN {X 0,Y 132.333,Z 279.326,A -85,B 0,C 180,E1 -30072.538,E2 -30072.538} C_VEL
LIN {X 0,Y 132.256,Z 281.409,A -85,B 0,C 180,E1 -30074.005,E2 -30074.005} C_VEL
LIN {X 0,Y 132.229,Z 288.338,A -85,B 0,C 180,E1 -30077.691,E2 -30077.691} C_VEL
LIN {X 0,Y 132.416,Z 289.583,A -85,B 0,C 180,E1 -30078.744,E2 -30078.744} C_VEL
LIN {X 0,Y 132.913,Z 291.812,A -85,B 0,C 180,E1 -30080.736,E2 -30080.736} C_VEL
LIN {X 0,Y 128.987,Z 321.934,A -85,B 0,C 180,E1 -30081.313,E2 -30081.313} C_VEL
LIN {X 0,Y 125.6,Z 337.318,A -85,B 0,C 180,E1 -30081.747,E2 -30081.747} C_VEL
LIN {X 0,Y 121.095,Z 351.806,A -85,B 0,C 180,E1 -30082.333,E2 -30082.333} C_VEL
LIN {X 0,Y 115.59,Z 365.476,A -85,B 0,C 180,E1 -30083.126,E2 -30083.126} C_VEL
LIN {X 0,Y 108.818,Z 378.944,A -85,B 0,C 180,E1 -30084.176,E2 -30084.176} C_VEL
LIN {X 0,Y 100.366,Z 392.687,A -85,B 0,C 180,E1 -30085.633,E2 -30085.633} C_VEL
LIN {X 0,Y 90.684,Z 405.686,A -85,B 0,C 180,E1 -30087.652,E2 -30087.652} C_VEL
LIN {X 0,Y 81.179,Z 416.461,A -85,B 0,C 180,E1 -30090.028,E2 -30090.028} C_VEL
LIN {X 0,Y 69.769,Z 427.459,A -85,B 0,C 180,E1 -30093.79,E2 -30093.79} C_VEL
LIN {X 0,Y 58.74,Z 436.586,A -85,B 0,C 180,E1 -30098.945,E2 -30098.945} C_VEL
LIN {X 0,Y 46.89,Z 445.121,A -85,B 0,C 180,E1 -30107.576,E2 -30107.576} C_VEL
LIN {X 0,Y 36.439,Z 451.997,A -85,B 0,C 180,E1 -30121.167,E2 -30121.167} C_VEL
LIN {X 0,Y 30.381,Z 456.161,A -85,B 0,C 180,E1 -30136.619,E2 -30136.619} C_VEL
LIN {X 0,Y 26.737,Z 459.608,A -85,B 0,C 180,E1 -30157.546,E2 -30157.546} C_VEL
LIN {X 0,Y 26.921,Z 462.265,A -85,B 0,C 180,E1 -30181.467,E2 -30181.467} C_VEL
LIN {X 0,Y 33.005,Z 464.736,A -85,B 0,C 180,E1 -30208.392,E2 -30208.392} C_VEL
LIN {X 0,Y 43.605,Z 465.925,A -85,B 0,C 180,E1 -30225.238,E2 -30225.238} C_VEL
LIN {X 0,Y 56.411,Z 465.825,A -85,B 0,C 180,E1 -30235.304,E2 -30235.304} C_VEL
LIN {X 0,Y 70.306,Z 464.416,A -85,B 0,C 180,E1 -30241.645,E2 -30241.645} C_VEL
LIN {X 0,Y 84.779,Z 461.658,A -85,B 0,C 180,E1 -30245.875,E2 -30245.875} C_VEL
LIN {X 0,Y 96.686,Z 458.385,A -85,B 0,C 180,E1 -30248.357,E2 -30248.357} C_VEL
LIN {X 0,Y 92.605,Z 459.679,A -85,B 0,C 180,E1 -30249.401,E2 -30249.401} C_VEL
LIN {X 0,Y 79.145,Z 463.137,A -85,B 0,C 180,E1 -30252.377,E2 -30252.377} C_VEL
LIN {X 0,Y 66.005,Z 465.47,A -85,B 0,C 180,E1 -30256.613,E2 -30256.613} C_VEL
LIN {X 0,Y 53.379,Z 466.731,A -85,B 0,C 180,E1 -30262.842,E2 -30262.842} C_VEL
LIN {X 0,Y 41.873,Z 466.875,A -85,B 0,C 180,E1 -30272.951,E2 -30272.951} C_VEL
LIN {X 0,Y 32.538,Z 465.945,A -85,B 0,C 180,E1 -30289.617,E2 -30289.617} C_VEL
LIN {X 0,Y 27.505,Z 463.938,A -85,B 0,C 180,E1 -30315.202,E2 -30315.202} C_VEL
LIN {X 0,Y 27.13,Z 462.495,A -85,B 0,C 180,E1 -30330.006,E2 -30330.006} C_VEL
LIN {X 0,Y 28.156,Z 459.597,A -85,B 0,C 180,E1 -30351.994,E2 -30351.994} C_VEL
LIN {X 0,Y 34.394,Z 454.524,A -85,B 0,C 180,E1 -30375.665,E2 -30375.665} C_VEL
LIN {X 0,Y 44.239,Z 447.991,A -85,B 0,C 180,E1 -30390.645,E2 -30390.645} C_VEL
LIN {X 0,Y 54.533,Z 440.795,A -85,B 0,C 180,E1 -30399.133,E2 -30399.133} C_VEL
LIN {X 0,Y 65.542,Z 432.164,A -85,B 0,C 180,E1 -30404.821,E2 -30404.821} C_VEL
LIN {X 0,Y 75.313,Z 423.357,A -85,B 0,C 180,E1 -30408.486,E2 -30408.486} C_VEL
LIN {X 0,Y 85.346,Z 412.931,A -85,B 0,C 180,E1 -30411.19,E2 -30411.19} C_VEL
LIN {X 0,Y 95.51,Z 400.443,A -85,B 0,C 180,E1 -30413.419,E2 -30413.419} C_VEL
LIN {X 0,Y 104.087,Z 387.918,A -85,B 0,C 180,E1 -30414.848,E2 -30414.848} C_VEL
LIN {X 0,Y 111.848,Z 374.202,A -85,B 0,C 180,E1 -30415.978,E2 -30415.978} C_VEL
LIN {X 0,Y 118.424,Z 359.792,A -85,B 0,C 180,E1 -30416.827,E2 -30416.827} C_VEL
LIN {X 0,Y 123.562,Z 345.435,A -85,B 0,C 180,E1 -30417.377,E2 -30417.377} C_VEL
LIN {X 0,Y 127.545,Z 330.212,A -85,B 0,C 180,E1 -30417.852,E2 -30417.852} C_VEL
LIN {X 0,Y 129.997,Z 316.11,A -85,B 0,C 180,E1 -30418.129,E2 -30418.129} C_VEL
LIN {X 0,Y 132.962,Z 292.017,A -85,B 0,C 180,E1 -30418.573,E2 -30418.573} C_VEL
LIN {X 0,Y 132.437,Z 289.402,A -85,B 0,C 180,E1 -30420.738,E2 -30420.738} C_VEL
LIN {X 0,Y 131.843,Z 286.613,A -85,B 0,C 180,E1 -30424.102,E2 -30424.102} C_VEL
LIN {X 0,Y 131.65,Z 285.377,A -85,B 0,C 180,E1 -30426.13,E2 -30426.13} C_VEL
LIN {X 0,Y 131.45,Z 285.381,A -85,B 0,C 180,E1 -30430.766,E2 -30430.766} C_VEL
LIN {X 0,Y 131.603,Z 285.872,A -85,B 0,C 180,E1 -30433.432,E2 -30433.432} C_VEL
LIN {X 0,Y 132.182,Z 288.663,A -85,B 0,C 180,E1 -30437.675,E2 -30437.675} C_VEL
LIN {X 0,Y 132.416,Z 289.583,A -85,B 0,C 180,E1 -30438.744,E2 -30438.744} C_VEL
LIN {X 0,Y 132.458,Z 291.133,A -85,B 0,C 180,E1 -30439.405,E2 -30439.405} C_VEL
LIN {X 0,Y 132.196,Z 294.003,A -85,B 0,C 180,E1 -30439.687,E2 -30439.687} C_VEL
LIN {X 0,Y 131.518,Z 298.432,A -85,B 0,C 180,E1 -30439.408,E2 -30439.408} C_VEL
LIN {X 0,Y 129.905,Z 307.482,A -85,B 0,C 180,E1 -30438.123,E2 -30438.123} C_VEL
LIN {X 0,Y 129.467,Z 310.611,A -85,B 0,C 180,E1 -30438.009,E2 -30438.009} C_VEL
LIN {X 0,Y 126.9,Z 326.674,A -85,B 0,C 180,E1 -30438.289,E2 -30438.289} C_VEL
LIN {X 0,Y 123.001,Z 342.213,A -85,B 0,C 180,E1 -30438.695,E2 -30438.695} C_VEL
LIN {X 0,Y 118.158,Z 356.227,A -85,B 0,C 180,E1 -30439.22,E2 -30439.22} C_VEL
LIN {X 0,Y 112.116,Z 369.917,A -85,B 0,C 180,E1 -30439.897,E2 -30439.897} C_VEL
LIN {X 0,Y 104.379,Z 384.046,A -85,B 0,C 180,E1 -30440.891,E2 -30440.891} C_VEL
LIN {X 0,Y 96.656,Z 395.699,A -85,B 0,C 180,E1 -30442.012,E2 -30442.012} C_VEL
LIN {X 0,Y 86.846,Z 408.11,A -85,B 0,C 180,E1 -30443.634,E2 -30443.634} C_VEL
LIN {X 0,Y 76.152,Z 419.461,A -85,B 0,C 180,E1 -30445.86,E2 -30445.86} C_VEL
LIN {X 0,Y 64.391,Z 429.98,A -85,B 0,C 180,E1 -30449.165,E2 -30449.165} C_VEL
LIN {X 0,Y 52.91,Z 438.702,A -85,B 0,C 180,E1 -30453.877,E2 -30453.877} C_VEL
LIN {X 0,Y 41.849,Z 445.961,A -85,B 0,C 180,E1 -30460.905,E2 -30460.905} C_VEL
LIN {X 0,Y 30.306,Z 452.702,A -85,B 0,C 180,E1 -30474.56,E2 -30474.56} C_VEL
LIN {X 0,Y 23.299,Z 456.812,A -85,B 0,C 180,E1 -30492.436,E2 -30492.436} C_VEL
LIN {X 0,Y 20.176,Z 459.118,A -85,B 0,C 180,E1 -30509.992,E2 -30509.992} C_VEL
LIN {X 0,Y 20.827,Z 462.747,A -85,B 0,C 180,E1 -30552.435,E2 -30552.435} C_VEL
LIN {X 0,Y 29.703,Z 465.102,A -85,B 0,C 180,E1 -30581.148,E2 -30581.148} C_VEL
LIN {X 0,Y 42.295,Z 466.174,A -85,B 0,C 180,E1 -30595.521,E2 -30595.521} C_VEL
LIN {X 0,Y 56.312,Z 465.952,A -85,B 0,C 180,E1 -30603.25,E2 -30603.25} C_VEL
LIN {X 0,Y 70.962,Z 464.421,A -85,B 0,C 180,E1 -30607.962,E2 -30607.962} C_VEL
LIN {X 0,Y 71.095,Z 464.423,A -85,B 0,C 180,E1 -30608.696,E2 -30608.696} C_VEL
LIN {X 0,Y 57.632,Z 466.111,A -85,B 0,C 180,E1 -30612.703,E2 -30612.703} C_VEL
LIN {X 0,Y 44.604,Z 466.742,A -85,B 0,C 180,E1 -30619.032,E2 -30619.032} C_VEL
LIN {X 0,Y 32.672,Z 466.264,A -85,B 0,C 180,E1 -30630.646,E2 -30630.646} C_VEL
LIN {X 0,Y 23.33,Z 464.698,A -85,B 0,C 180,E1 -30652.96,E2 -30652.96} C_VEL
LIN {X 0,Y 20.7,Z 463.503,A -85,B 0,C 180,E1 -30670.161,E2 -30670.161} C_VEL
LIN {X 0,Y 20.013,Z 462.006,A -85,B 0,C 180,E1 -30690.008,E2 -30690.008} C_VEL
LIN {X 0,Y 21.696,Z 459.051,A -85,B 0,C 180,E1 -30719.08,E2 -30719.08} C_VEL
LIN {X 0,Y 29.823,Z 453.857,A -85,B 0,C 180,E1 -30745.579,E2 -30745.579} C_VEL
LIN {X 0,Y 40.741,Z 447.464,A -85,B 0,C 180,E1 -30759.047,E2 -30759.047} C_VEL
LIN {X 0,Y 52.405,Z 439.862,A -85,B 0,C 180,E1 -30766.493,E2 -30766.493} C_VEL
LIN {X 0,Y 64.033,Z 431.072,A -85,B 0,C 180,E1 -30771.06,E2 -30771.06} C_VEL
LIN {X 0,Y 75.918,Z 420.414,A -85,B 0,C 180,E1 -30774.384,E2 -30774.384} C_VEL
LIN {X 0,Y 86.271,Z 409.491,A -85,B 0,C 180,E1 -30776.355,E2 -30776.355} C_VEL
LIN {X 0,Y 95.825,Z 397.506,A -85,B 0,C 180,E1 -30777.879,E2 -30777.879} C_VEL
LIN {X 0,Y 103.688,Z 385.876,A -85,B 0,C 180,E1 -30778.824,E2 -30778.824} C_VEL
LIN {X 0,Y 110.697,Z 373.509,A -85,B 0,C 180,E1 -30779.586,E2 -30779.586} C_VEL
LIN {X 0,Y 117.26,Z 359.224,A -85,B 0,C 180,E1 -30780.228,E2 -30780.228} C_VEL
LIN {X 0,Y 122.433,Z 344.842,A -85,B 0,C 180,E1 -30780.645,E2 -30780.645} C_VEL
LIN {X 0,Y 126.527,Z 329.193,A -85,B 0,C 180,E1 -30781.009,E2 -30781.009} C_VEL
LIN {X 0,Y 128.957,Z 314.947,A -85,B 0,C 180,E1 -30781.261,E2 -30781.261} C_VEL
LIN {X 0,Y 131.29,Z 296.139,A -85,B 0,C 180,E1 -30781.58,E2 -30781.58} C_VEL
LIN {X 0,Y 130.777,Z 293.149,A -85,B 0,C 180,E1 -30785.328,E2 -30785.328} C_VEL
LIN {X 0,Y 130.662,Z 292.35,A -85,B 0,C 180,E1 -30786.998,E2 -30786.998} C_VEL
LIN {X 0,Y 130.564,Z 292.482,A -85,B 0,C 180,E1 -30791.241,E2 -30791.241} C_VEL
LIN {X 0,Y 130.649,Z 292.91,A -85,B 0,C 180,E1 -30792.979,E2 -30792.979} C_VEL
LIN {X 0,Y 131.072,Z 295.397,A -85,B 0,C 180,E1 -30796.824,E2 -30796.824} C_VEL
LIN {X 0,Y 131.238,Z 296.172,A -85,B 0,C 180,E1 -30797.742,E2 -30797.742} C_VEL
LIN {X 0,Y 129.467,Z 310.611,A -85,B 0,C 180,E1 -30798.009,E2 -30798.009} C_VEL
LIN {X 0,Y 128.592,Z 316.436,A -85,B 0,C 180,E1 -30797.812,E2 -30797.812} C_VEL
LIN {X 0,Y 126.611,Z 325.828,A -85,B 0,C 180,E1 -30796.68,E2 -30796.68} C_VEL
LIN {X 0,Y 124.211,Z 335.122,A -85,B 0,C 180,E1 -30795.529,E2 -30795.529} C_VEL
LIN {X 0,Y 123.137,Z 338.899,A -85,B 0,C 180,E1 -30795.347,E2 -30795.347} C_VEL
LIN {X 0,Y 122.58,Z 340.794,A -85,B 0,C 180,E1 -30795.372,E2 -30795.372} C_VEL
LIN {X 0,Y 117.748,Z 355.042,A -85,B 0,C 180,E1 -30795.746,E2 -30795.746} C_VEL
LIN {X 0,Y 111.646,Z 369.01,A -85,B 0,C 180,E1 -30796.26,E2 -30796.26} C_VEL
LIN {X 0,Y 103.793,Z 383.36,A -85,B 0,C 180,E1 -30796.97,E2 -30796.97} C_VEL
LIN {X 0,Y 95.945,Z 395.172,A -85,B 0,C 180,E1 -30797.77,E2 -30797.77} C_VEL
LIN {X 0,Y 87.405,Z 406.077,A -85,B 0,C 180,E1 -30798.764,E2 -30798.764} C_VEL
LIN {X 0,Y 76.784,Z 417.497,A -85,B 0,C 180,E1 -30800.246,E2 -30800.246} C_VEL
LIN {X 0,Y 66.393,Z 426.963,A -85,B 0,C 180,E1 -30802.138,E2 -30802.138} C_VEL
LIN {X 0,Y 54.383,Z 436.226,A -85,B 0,C 180,E1 -30805.22,E2 -30805.22} C_VEL
LIN {X 0,Y 42.05,Z 444.223,A -85,B 0,C 180,E1 -30810.098,E2 -30810.098} C_VEL
LIN {X 0,Y 31.007,Z 450.297,A -85,B 0,C 180,E1 -30817.496,E2 -30817.496} C_VEL
LIN {X 0,Y 19.001,Z 456.165,A -85,B 0,C 180,E1 -30836.293,E2 -30836.293} C_VEL
LIN {X 0,Y 12.705,Z 459.714,A -85,B 0,C 180,E1 -30869.987,E2 -30869.987} C_VEL
LIN {X 0,Y 16.067,Z 463.229,A -85,B 0,C 180,E1 -30931.003,E2 -30931.003} C_VEL
LIN {X 0,Y 28.172,Z 465.47,A -85,B 0,C 180,E1 -30956.19,E2 -30956.19} C_VEL
LIN {X 0,Y 42.403,Z 466.423,A -85,B 0,C 180,E1 -30966.07,E2 -30966.07} C_VEL
LIN {X 0,Y 44.782,Z 466.529,A -85,B 0,C 180,E1 -30969.025,E2 -30969.025} C_VEL
LIN {X 0,Y 29.667,Z 465.984,A -85,B 0,C 180,E1 -30978.649,E2 -30978.649} C_VEL
LIN {X 0,Y 18.157,Z 464.316,A -85,B 0,C 180,E1 -30999.287,E2 -30999.287} C_VEL
LIN {X 0,Y 14.219,Z 463.069,A -85,B 0,C 180,E1 -31020.392,E2 -31020.392} C_VEL
LIN {X 0,Y 12.911,Z 461.518,A -85,B 0,C 180,E1 -31050.012,E2 -31050.012} C_VEL
LIN {X 0,Y 15.821,Z 458.503,A -85,B 0,C 180,E1 -31091.797,E2 -31091.797} C_VEL
LIN {X 0,Y 26.44,Z 453.191,A -85,B 0,C 180,E1 -31118.505,E2 -31118.505} C_VEL
LIN {X 0,Y 39.308,Z 446.359,A -85,B 0,C 180,E1 -31129.363,E2 -31129.363} C_VEL
LIN {X 0,Y 52.921,Z 437.783,A -85,B 0,C 180,E1 -31134.914,E2 -31134.914} C_VEL
LIN {X 0,Y 65.054,Z 428.586,A -85,B 0,C 180,E1 -31137.934,E2 -31137.934} C_VEL
LIN {X 0,Y 77.108,Z 417.675,A -85,B 0,C 180,E1 -31140.002,E2 -31140.002} C_VEL
LIN {X 0,Y 87.878,Z 405.985,A -85,B 0,C 180,E1 -31141.373,E2 -31141.373} C_VEL
LIN {X 0,Y 97.596,Z 393.347,A -85,B 0,C 180,E1 -31142.307,E2 -31142.307} C_VEL
LIN {X 0,Y 105.563,Z 380.886,A -85,B 0,C 180,E1 -31142.953,E2 -31142.953} C_VEL
LIN {X 0,Y 113.191,Z 366.279,A -85,B 0,C 180,E1 -31143.473,E2 -31143.473} C_VEL
LIN {X 0,Y 119.311,Z 351.378,A -85,B 0,C 180,E1 -31143.814,E2 -31143.814} C_VEL
LIN {X 0,Y 123.98,Z 336.215,A -85,B 0,C 180,E1 -31144.131,E2 -31144.131} C_VEL
LIN {X 0,Y 127.302,Z 320.645,A -85,B 0,C 180,E1 -31144.285,E2 -31144.285} C_VEL
LIN {X 0,Y 129.899,Z 301.046,A -85,B 0,C 180,E1 -31144.592,E2 -31144.592} C_VEL
LIN {X 0,Y 129.76,Z 299.391,A -85,B 0,C 180,E1 -31147.047,E2 -31147.047} C_VEL
LIN {X 0,Y 129.669,Z 299.542,A -85,B 0,C 180,E1 -31151.319,E2 -31151.319} C_VEL
LIN {X 0,Y 129.744,Z 300.389,A -85,B 0,C 180,E1 -31153.37,E2 -31153.37} C_VEL
LIN {X 0,Y 129.858,Z 301.137,A -85,B 0,C 180,E1 -31154.708,E2 -31154.708} C_VEL
LIN {X 0,Y 126.749,Z 323.321,A -85,B 0,C 180,E1 -31155.056,E2 -31155.056} C_VEL
LIN {X 0,Y 123.416,Z 337.886,A -85,B 0,C 180,E1 -31155.302,E2 -31155.302} C_VEL
LIN {X 0,Y 122.58,Z 340.794,A -85,B 0,C 180,E1 -31155.372,E2 -31155.372} C_VEL
LIN {X 0,Y 121.433,Z 344.562,A -85,B 0,C 180,E1 -31155.301,E2 -31155.301} C_VEL
LIN {X 0,Y 118.797,Z 351.87,A -85,B 0,C 180,E1 -31154.573,E2 -31154.573} C_VEL
LIN {X 0,Y 113.482,Z 364.251,A -85,B 0,C 180,E1 -31152.828,E2 -31152.828} C_VEL
LIN {X 0,Y 110.923,Z 369.524,A -85,B 0,C 180,E1 -31152.632,E2 -31152.632} C_VEL
LIN {X 0,Y 103.698,Z 382.672,A -85,B 0,C 180,E1 -31153.023,E2 -31153.023} C_VEL
LIN {X 0,Y 95.766,Z 394.645,A -85,B 0,C 180,E1 -31153.49,E2 -31153.49} C_VEL
LIN {X 0,Y 86.246,Z 406.661,A -85,B 0,C 180,E1 -31154.152,E2 -31154.152} C_VEL
LIN {X 0,Y 76.374,Z 417.176,A -85,B 0,C 180,E1 -31154.926,E2 -31154.926} C_VEL
LIN {X 0,Y 64.033,Z 428.151,A -85,B 0,C 180,E1 -31156.177,E2 -31156.177} C_VEL
LIN {X 0,Y 51.719,Z 437.264,A -85,B 0,C 180,E1 -31157.961,E2 -31157.961} C_VEL
LIN {X 0,Y 39.898,Z 444.571,A -85,B 0,C 180,E1 -31160.632,E2 -31160.632} C_VEL
LIN {X 0,Y 27.22,Z 451.069,A -85,B 0,C 180,E1 -31165.34,E2 -31165.34} C_VEL
LIN {X 0,Y 16.892,Z 455.521,A -85,B 0,C 180,E1 -31173.665,E2 -31173.665} C_VEL
LIN {X 0,Y 8.934,Z 458.54,A -85,B 0,C 180,E1 -31191.905,E2 -31191.905} C_VEL
LIN {X 0,Y 7.558,Z 462.138,A -85,B 0,C 180,E1 -31298.355,E2 -31298.355} C_VEL
LIN {X 0,Y 14.408,Z 463.754,A -85,B 0,C 180,E1 -31319.989,E2 -31319.989} C_VEL
LIN {X 0,Y 21.27,Z 464.927,A -85,B 0,C 180,E1 -31327.647,E2 -31327.647} C_VEL
LIN {X 0,Y 21.342,Z 464.951,A -85,B 0,C 180,E1 -31328.965,E2 -31328.965} C_VEL
LIN {X 0,Y 8.762,Z 462.634,A -85,B 0,C 180,E1 -31356.702,E2 -31356.702} C_VEL
LIN {X 0,Y 5.798,Z 461.03,A -85,B 0,C 180,E1 -31410.028,E2 -31410.028} C_VEL
LIN {X 0,Y 11.519,Z 457.942,A -85,B 0,C 180,E1 -31476.263,E2 -31476.263} C_VEL
LIN {X 0,Y 24.727,Z 452.521,A -85,B 0,C 180,E1 -31494.212,E2 -31494.212} C_VEL
LIN {X 0,Y 39.108,Z 445.296,A -85,B 0,C 180,E1 -31500.004,E2 -31500.004} C_VEL
LIN {X 0,Y 52.772,Z 436.803,A -85,B 0,C 180,E1 -31502.713,E2 -31502.713} C_VEL
LIN {X 0,Y 65.195,Z 427.447,A -85,B 0,C 180,E1 -31504.294,E2 -31504.294} C_VEL
LIN {X 0,Y 76.412,Z 417.363,A -85,B 0,C 180,E1 -31505.279,E2 -31505.279} C_VEL
LIN {X 0,Y 87.455,Z 405.473,A -85,B 0,C 180,E1 -31506.008,E2 -31506.008} C_VEL
LIN {X 0,Y 97.259,Z 392.768,A -85,B 0,C 180,E1 -31506.478,E2 -31506.478} C_VEL
LIN {X 0,Y 105.287,Z 380.254,A -85,B 0,C 180,E1 -31506.806,E2 -31506.806} C_VEL
LIN {X 0,Y 112.49,Z 366.539,A -85,B 0,C 180,E1 -31507.062,E2 -31507.062} C_VEL
LIN {X 0,Y 118.662,Z 351.732,A -85,B 0,C 180,E1 -31507.221,E2 -31507.221} C_VEL
LIN {X 0,Y 123.475,Z 336.339,A -85,B 0,C 180,E1 -31507.412,E2 -31507.412} C_VEL
LIN {X 0,Y 126.824,Z 320.886,A -85,B 0,C 180,E1 -31507.476,E2 -31507.476} C_VEL
LIN {X 0,Y 128.813,Z 306.407,A -85,B 0,C 180,E1 -31507.725,E2 -31507.725} C_VEL
LIN {X 0,Y 128.779,Z 306.668,A -85,B 0,C 180,E1 -31511.638,E2 -31511.638} C_VEL
LIN {X 0,Y 126.005,Z 325.06,A -85,B 0,C 180,E1 -31511.871,E2 -31511.871} C_VEL
LIN {X 0,Y 122.156,Z 340.816,A -85,B 0,C 180,E1 -31512.064,E2 -31512.064} C_VEL
LIN {X 0,Y 116.9,Z 356.098,A -85,B 0,C 180,E1 -31512.32,E2 -31512.32} C_VEL
LIN {X 0,Y 110.923,Z 369.524,A -85,B 0,C 180,E1 -31512.632,E2 -31512.632} C_VEL
LIN {X 0,Y 110.714,Z 370.417,A -85,B 0,C 180,E1 -31512.644,E2 -31512.644} C_VEL
LIN {X 0,Y 110.714,Z 600,A -85,B 0,C 180,E1 -31512.644,E2 -31512.644} C_VEL
LIN {X 0,Y 110.714,Z 600,A -85,B 0,C 180,E1 -31512.644,E2 -31512.644}

QRS_NEXT_CUT()

QRS_NEXT()
QRS_HOME()

END
